							ExtVelocity[axisIdx]:= (newPos - OldPosition[axisIdx]) / (UDINT_TO_LREAL(_TaskInfo[1].CycleTime) / 10000000);
							OldPosition[axisIdx]:= newPos;
							ExtAcceleration :=  (ExtVelocity[axisIdx] - OldVelocity[axisIdx]) / (UDINT_TO_LREAL(_TaskInfo[1].CycleTime) / 10000000);
							OldVelocity[axisIdx]:= ExtVelocity[axisIdx];
							ExtDirection := SEL(newPos >= OldPosition[axisIdx], -1, 1);

							MC_ExtSetPointGenFeed(
								Position := newPos,
								Velocity := ExtVelocity[axisIdx],
								Acceleration := ExtAcceleration,
								Direction := ExtDirection,
								Axis := Axis[axisIdx].Axis);

						(*一般軸處理*)
						ELSE
							ExtVelocity[axisIdx]:= (TableOffsetPos[axisIdx] - OldPosition[axisIdx]) / (UDINT_TO_LREAL(_TaskInfo[1].CycleTime) / 10000000);
							OldPosition[axisIdx]:= TableOffsetPos[axisIdx];
							ExtAcceleration :=  (ExtVelocity[axisIdx] - OldVelocity[axisIdx]) / (UDINT_TO_LREAL(_TaskInfo[1].CycleTime) / 10000000);
							OldVelocity[axisIdx]:= ExtVelocity[axisIdx];
							ExtDirection := SEL(TableOffsetPos[axisIdx] >= OldPosition[axisIdx], -1, 1);
							//ExtDirection := SEL(TableOffsetPos[axisIdx] >= OldPosition[axisIdx], -1, 1);

							MC_ExtSetPointGenFeed(
								Position := TableOffsetPos[axisIdx],
								Velocity := ExtVelocity[axisIdx],
								Acceleration := ExtAcceleration,
								Direction := ExtDirection,
								Axis := Axis[axisIdx].Axis);
						END_IF
					END_IF
				END_FOR

				(* 目前送線動作結束 改idx*)
				IF AxisIsOn[FeederNo]
				AND CurrentTableIdx = FeederEndIdx[FeederIdx] + 1
				AND FeederEndIdx[FeederIdx] <> 0 THEN		

					FeederIdx := FeederIdx + 1;
					TouchOpenNo := 0;
					
				END_IF

				(* 探針動作結束 初始化 *)
				FOR touchIdx := 1 TO TouchNo DO

					IF CurrentTableIdx = TouchConfig[touchIdx].EndIdx[TouchConfigIdx[touchIdx]]
					AND TouchConfig[touchIdx].EndIdx[TouchConfigIdx[touchIdx]] <> 0 THEN
						IsTouch := FALSE;
						IsPreTouch := FALSE;
						TouchConfigIdx[touchIdx] := TouchConfigIdx[touchIdx] + 1;
					END_IF

					IF TouchConfigIdx[touchIdx] > 0 THEN
						IF CurrentTableIdx = TouchConfig[touchIdx].EndIdx[TouchConfigIdx[touchIdx] - 1] + 1
						AND TouchConfig[touchIdx].EndIdx[TouchConfigIdx[touchIdx] - 1] <> 0 THEN
							TouchMiss := FALSE;
						END_IF
					END_IF

				END_FOR

				(* 下一個探針動作的開始 先檢查是否探針前失誤 *)
								TouchPreCheck();

								NextCycleIdx();
				
								
				NextSubProgram();

			END_IF
	END_CASE

END_IF

ACTION AirFunc:

(*----------------Air----------------1,2,7,8是探針汽缸*)
(*非測試編輯時跑表*)
IF NOT (Inputstate.VRSwitch = FALSE AND State = ENUMSTATE.S_TEST) THEN
	FOR airIdx := 1 TO AirNo DO
		IF  airIdx <> 1 
		AND airIdx <> 2 
		AND airIdx <> 7
		AND airIdx <> 8 
		THEN
			AirIsOpen[airIdx] := AirTable[airIdx, CurrentTableIdx];
		END_IF
	END_FOR
END_IF
END_ACTION

ACTION CtrlSpeed:
IF Inputstate.ExFeederError
OR (IOSwitch.SaftyEnable AND 
        (Inputstate.SafetyError OR Inputstate.SafetyError1 OR Inputstate.SafetyError2 OR Inputstate.SafetyError3 OR Inputstate.SafetyError4) 
    ) 
THEN
    SpeedDownTo0 := TRUE;
    IF SpeedUPToOverride THEN
	    SpeedUPToOverride := FALSE;
        SpeedCtrlAccTimer(IN:=FALSE);
    END_IF
END_IF


IF lState <> State THEN
    lState := State;
    SpeedChanged := TRUE;
END_IF

IF SpeedUPToOverride THEN
	(*Reset Timer*)
	IF SpeedDownTo0 THEN
		SpeedDownTo0 := FALSE;
		SpeedCtrlDecTimer(IN:=FALSE);
	END_IF
    SpeedCtrlAccTimer(IN:=TRUE , PT:=SpeedAccDccTime , Q=> , ET=> );
    Speed        := Override * TIME_TO_REAL(SpeedCtrlAccTimer.ET) / TIME_TO_REAL(SpeedCtrlAccTimer.PT); (* 0 -> 1 *)
    IF SpeedCtrlAccTimer.Q THEN
        SpeedCtrlAccTimer(IN:=FALSE);
        SpeedUPToOverride := FALSE;
    END_IF
ELSIF SpeedDownTo0 THEN
    SpeedCtrlDecTimer(IN:=TRUE , PT:=SpeedAccDccTime , Q=> , ET=> );
    Speed        := Override * ( TIME_TO_REAL(SpeedCtrlDecTimer.PT) - TIME_TO_REAL(SpeedCtrlDecTimer.ET) ) / TIME_TO_REAL(SpeedCtrlDecTimer.PT); (* 1 -> 0 *)
ELSE
    IF SpeedChanged THEN
        IF LREAL_TO_DINT(Speed * 1000.0/100.0) = LREAL_TO_DINT(Override * 1000.0/100.0) THEN
            SpeedChanged := FALSE;
        ELSIF Speed < Override THEN
            Speed := Speed + 100.0/1000.0; (* 0->100% 用 1000ms *)
        ELSIF Speed > Override THEN
            Speed := Speed - 100.0/1000.0; (* 0->100% 用 1000ms *)
        END_IF
    ELSE
        Speed := Override;
    END_IF
END_IF
END_ACTION

ACTION EnableExtSetPoint:
	

FOR axisIdx := 1 TO No DO
	IF AxisIsOn[axisIdx] THEN
		Axis[axisIdx].EnableSetPointGenerator
		(
			Execute := TRUE,
			Position := Axis[axisIdx].ActPos,
			PositionType := POSITIONTYPE_ABSOLUTE,
			Axis :=  Axis[axisIdx].Axis
		);
	END_IF
END_FOR
ProduceState := S_WaitExtSetPoint;
END_ACTION

ACTION ExFeederFunc:

(*-------ExFeederSpeedUp------*)
IF State = ENUMSTATE.S_AUTO THEN
	ExFeederSpeedUp := ExFSpdUpTable[CurrentTableIdx];
END_IF
END_ACTION

ACTION FeederPosSetting:

FNeedHoldPos(
	IsTouch:= IsTouch,
	IsPreTouch := IsPreTouch,
	CurrentIdx:= CurrentTableIdx,
	FeederIdx	:= FeederIdx,
	FeederStartIdx:= FeederStartIdx,
	FeederEndIdx:=  FeederEndIdx,
	TouchConfig	    := TouchConfig,
	TouchConfigIdx := TouchConfigIdx,
 );

(* 計算位置 *)
IF FlashModeOn THEN

	IF(CurrentTableIdx = RepeatA) THEN
		(*閃電模式下，在A點是新的彈簧開始，根據offset進來次數不一定只會一次*)
		IF JumpFirstTime THEN
			JumpFirstTime := FALSE;
			Feeder.StillPos 	 := AxisTable1[axisIdx, FeederStartIdx[FeederIdx]] ;
			IF FNeedHoldPos.Yes = FALSE THEN
				Feeder.BasePos 	 := Feeder.CurPos - ( AxisTable1[axisIdx, RepeatA - 1] + ( AxisTable1[axisIdx, RepeatA] - AxisTable1[axisIdx, RepeatA - 1] ) * LastTableOffset );
			END_IF
		END_IF	
	ELSIF (CurrentTableIdx = JumpTiming) THEN
		IF JumpFirstTime THEN
			JumpFirstTime := FALSE;
			IF FNeedHoldPos.Yes = FALSE THEN
				Feeder.BasePos := Feeder.CurPos - ( AxisTable1[axisIdx, JumpTiming - 1] + ( AxisTable1[axisIdx, JumpTiming] - AxisTable1[axisIdx, JumpTiming - 1] ) * LastTableOffset );
			END_IF	
		END_IF
	END_IF

ELSIF CurrentTableIdx = G5Config[G5Status.CurIdx].ATime THEN

	IF G5Status.JumpFirstTime THEN
		G5Status.JumpFirstTime := FALSE;
		Feeder.StillPos 	 := AxisTable1[axisIdx, FeederStartIdx[FeederIdx]] ;	
		IF FNeedHoldPos.Yes = FALSE THEN
			Feeder.BasePos 	 := Feeder.CurPos - ( AxisTable1[axisIdx, CurrentTableIdx ]  );
		END_IF
	END_IF
	
END_IF

FSetCurPos();
END_ACTION

ACTION FeederVelAccSetting:
FNeedHoldPos(
	IsTouch:= IsTouch,
	IsPreTouch := IsPreTouch,
	CurrentIdx:= CurrentTableIdx,
	FeederIdx	:= FeederIdx,
	FeederStartIdx:= FeederStartIdx,
	FeederEndIdx:=  FeederEndIdx,
	TouchConfig	    := TouchConfig,
	TouchConfigIdx := TouchConfigIdx,
);
	
(*計算速度,加速度,方向*)
IF FNeedHoldPos.Yes THEN
	ExtVelocity[axisIdx]:= 0;
ELSE
	ExtVelocity[axisIdx]:= (Feeder.CurPos - OldPosition[axisIdx]) / (UDINT_TO_LREAL(_TaskInfo[1].CycleTime) / 10000000);
END_IF
OldPosition[axisIdx]:= Feeder.CurPos;
ExtDirection := SEL(Feeder.CurPos >= OldPosition[axisIdx], -1, 1);
ExtAcceleration :=  (ExtVelocity[axisIdx] - OldVelocity[axisIdx]) / (UDINT_TO_LREAL(_TaskInfo[1].CycleTime) / 10000000);
OldVelocity[axisIdx]:= ExtVelocity[axisIdx];
END_ACTION

ACTION FillAxisTable:
IF AxisTableBuf.OK THEN
	FOR axisIdx := 1 TO No DO
		FOR Idx := 0 TO 1999  DO
			AxisTable1[axisIdx, idx + SendOffset] := AxisTableBuf.Table[axisIdx, idx];
		END_FOR
	END_FOR
	SendOffset := SendOffset + 2000;
	AxisTableBuf.OK := FALSE;
	IF SendOffset >= TotalTimeByMs THEN
		SendOffset := 0;
		ProduceState := S_FillIOTable;
	END_IF
END_IF
IsGetTableBuf :=AxisTableBuf.OK;
END_ACTION

ACTION FillIOTable:

IsGetTableBuf := FALSE;
ReceiveAllBuf := TRUE;
IF TouchTableBuf.OK THEN
	TouchTableBuf.OK := FALSE;
	FOR touchIdx := 1 TO TouchNo DO
		FOR Idx := 0 TO 1999  DO
			TouchTable[touchIdx, idx + SendOffset] := TouchTableBuf.Table[touchIdx, idx];
		END_FOR
	END_FOR
	TouchTableFill := TRUE;
END_IF
IsGetTableBuf := IsGetTableBuf OR TouchTableFill;
ReceiveAllBuf := ReceiveAllBuf AND TouchTableFill;

IF AirTableBuf.OK THEN
	AirTableBuf.OK := FALSE;
	FOR airIdx := 1 TO AirNo DO
		FOR Idx := 0 TO 1999  DO
			AirTable[airIdx, idx + SendOffset] := AirTableBuf.Table[airIdx, idx];
		END_FOR
	END_FOR
	AirTableFill := TRUE;
END_IF
IsGetTableBuf := IsGetTableBuf OR AirTableFill;
ReceiveAllBuf := ReceiveAllBuf AND AirTableFill;

IF ExFSpdUpTableBuf.OK THEN
	ExFSpdUpTableBuf.OK := FALSE;
	FOR Idx := 0 TO 1999  DO
		ExFSpdUpTable[idx + SendOffset] := ExFSpdUpTableBuf.Table[idx];
	END_FOR
	ExFSpdUpTableFill := TRUE;
END_IF
IsGetTableBuf := IsGetTableBuf OR ExFSpdUpTableFill;
ReceiveAllBuf := ReceiveAllBuf AND ExFSpdUpTableFill;

IF ReceiveAllBuf THEN
	TouchTableFill := FALSE;
	AirTableFill := FALSE;
	ExFSpdUpTableFill := FALSE;
	SendOffset := SendOffset + 2000;
	IF SendOffset >= TotalTimeByMs THEN
		SendOffset := 0;
		ProduceState := S_FillSubTable;
	END_IF
END_IF
END_ACTION

ACTION FillSubIOTable:
IsGetTableBuf := FALSE;
IF SubProgramConfig[getSubNo].TotalTableSIze = 0 THEN
	ProduceState := S_FillTouchAdjustTable;
ELSE
    IF AirTableBuf.OK THEN
        FOR airIdx := 1 TO AirNo DO
            FOR Idx := 0 TO 1999  DO
                SubProgramTable[getSubNo].airTable[airIdx, idx + SendOffset] := AirTableBuf.Table[airIdx, idx];
            END_FOR
        END_FOR
        SendOffset := SendOffset + 2000;
        AirTableBuf.OK := FALSE;
        IF SendOffset >= SubProgramConfig[getSubNo].TotalTableSize THEN
            getSubNo := getSubNo + 1;
            SendOffset := 0;
        END_IF
    END_IF
    IsGetTableBuf := AirTableBuf.OK;
END_IF
END_ACTION

ACTION FillSubTable:

IsGetTableBuf := FALSE;
IF SubProgramConfig[getSubNo].TotalTableSIze = 0 THEN
	getSubNo := 1;
	ProduceState := S_FillSubIOTable;
ELSE
	IF AxisTableBuf.OK THEN
		FOR axisIdx := 1 TO No DO
			FOR Idx := 0 TO 1999  DO
				SubProgramTable[getSubNo].AxisTable[axisIdx, idx + SendOffset] := AxisTableBuf.Table[axisIdx, idx];
			END_FOR
		END_FOR
		SendOffset := SendOffset + 2000;
		AxisTableBuf.OK := FALSE;
		IF SendOffset >= SubProgramConfig[getSubNo].TotalTableSize THEN
			getSubNo := getSubNo + 1;
			SendOffset := 0;
		END_IF
	END_IF
	IsGetTableBuf := AxisTableBuf.OK;
END_IF
END_ACTION

ACTION FillTouchAdjustTable:
IsGetTableBuf := FALSE;
IF AxisTableBuf.OK THEN
    FOR axisIdx := 1 TO TouchAdjustNo DO
        IF TouchAdjustConfig[axisIdx].Enable THEN
            FOR idx := 0 TO 1999  DO
                TouchAdjustTable[axisIdx, idx + SendOffset] := AxisTableBuf.Table[axisIdx, idx];
            END_FOR
        END_IF        
    END_FOR
    SendOffset := SendOffset + 2000;
    AxisTableBuf.OK := FALSE;
    IF SendOffset >= TotalTimeByMs THEN
        SendOffset := 0;
        ProduceState := S_EnableExtSetPoint;
    END_IF
END_IF
IsGetTableBuf := AxisTableBuf.OK;
END_ACTION

ACTION FSetCurPos:

IF FNeedHoldPos.Yes THEN
	Feeder.CurPos := Feeder.BasePos + Feeder.TouchPos;
ELSE
	Feeder.CurPos := Feeder.BasePos + TableOffsetPos[axisIdx];
END_IF
END_ACTION

ACTION Initial:


FOR axisIdx:=1 TO No DO
	(*Set的最後一個點非0的時候沒清會爆衝*)
	Axis[axisIdx].Axis.PlcToNc.ExtSetPos := Axis[axisIdx].ActPos;
	Axis[axisIdx].EnableSetPointGenerator.Execute := FALSE;
	TableOffsetPos[axisIdx] := Axis[axisIdx].ActPos;
	OldPosition[axisIdx] := Axis[axisIdx].ActPos;
	OldVelocity[axisIdx] := 0;
	IsExtSetPointDone[axisIdx]:=FALSE;
	ModuloBase[axisIdx]  := Axis[axisIdx].ActPos;
END_FOR

ProFirstTime			:= FALSE;
Idx0FirstTime			:= TRUE;
ProduceState			:= S_FillAxisTable;
StartProNum				:= ProduceCurNum;
ProduceTimer			:= 0;
PPM						:= 0;
PPMCal(Clear := TRUE);
SpeedDownTo0			:= FALSE;
SpeedUPToOverride		:= FALSE;
SpeedCtrlAccTimer(IN:=FALSE);
SpeedCtrlDecTimer(IN:=FALSE);

JumpFirstTime		:= TRUE;

(*Send Table*)
getSubNo			:= 1;
SendOffset			:= 0;
TouchTableFill 		:= FALSE;
AirTableFill 			:= FALSE;
ExFSpdUpTableFill 	:= FALSE;

(*Index*)
CurrentTableIdx		:= 0;
CurrentTableOffset	:= 0;
LastTableOffset		:= 0;

(*IO*)
FOR touchIdx := 1 TO TouchNo DO
	TouchDist[touchIdx] 	 := 0;
	TouchConfigIdx[touchIdx] := 0;
	PreTouchShow[touchIdx]   := FALSE;
	ThisTurnTouchMissShow[touchIdx] := FALSE;
END_FOR
IsTouch				:= FALSE;
IsPreTouch			:= FALSE;
TouchOpenNo		:= 0;
TouchMiss			:= FALSE;
TouchBeforeStart		:= FALSE;
TouchMissNum		:= 0;
ThisTurnTouchMiss	:= FALSE;
IsOverUpBound		:= FALSE;
IsBelowDownBound	:= FALSE;
FeederIdx			:= 0;
Feeder.CurPos		:= Axis[FeederNo].Axis.NcToPlc.SetPos;
Feeder.BasePos	:= 0;
Feeder.StillPos		:= 0;
Feeder.TouchPos		:= 0;

AxisTableBuf.OK		:= FALSE;
TouchTableBuf.OK	:= FALSE;
AirTableBuf.OK		:= FALSE;
ExFSpdUpTableBuf.OK:= FALSE;

FOR TouchAdjustIdx := 1 TO TouchAdjustNo DO
	AdjustCounter[TouchAdjustIdx] := 0;
	AdjustCounterBuf[TouchAdjustIdx] := 0;
END_FOR

RunSubProgram		:= FALSE;
SubInFirstTime		:= TRUE;
RunSubNo			:=1;
SubTableIdx			:=0;
SubTableOffset		:=0;

(*油初始先開*)
FirstAutoRun := TRUE;

(*G5*)
G5Status.ATimeFIdx	   := 0;
G5Status.CurIdx		   := 1;
G5Status.CurTimes	   := 0;
G5Status.JumpFirstTime := FALSE;

lState	:= State;
SpeedChanged := FALSE;
END_ACTION

ACTION ModuloTurnsPlus1:
FOR axisIdx := 1 TO No DO
	IF AxesUseModulo[axisIdx] THEN
		AxesModuloTurns[axisIdx] := AxesModuloTurns[axisIdx] +  LREAL_TO_DINT( AxesModuloOGrad[axisIdx]) / AxesGradPerTurn[axisIdx];				
	END_IF
END_FOR
END_ACTION

ACTION NextCycleIdx:

(*探針失誤1次 設定也是一次 則 先暫停 => CurrentTableOffset 不變*)
IF TouchMissStop = FALSE THEN
	LastTableOffset := CurrentTableOffset;
	CurrentTableOffset := CurrentTableOffset + Speed/100;
END_IF

(*CurrentTableIdx增加的時候*)
IF CurrentTableOffset >= 1 THEN
	CurrentTableOffset := CurrentTableOffset - 1;
	(*閃電模式*)
	IF FlashModeOn THEN
		(*RepeatA*)
		IF CurrentTableIdx = RepeatA THEN
			(*紀錄RepeatA時的FeederIdx給跳回來時設定*)
			RepeatA_FeederIdx 	:= FeederIdx;
			FOR touchIdx := 1 TO TouchNo DO
				RepeatA_TouchConfigIdx[touchIdx] := TouchConfigIdx[touchIdx];
			END_FOR
			CurrentTableIdx 	:= CurrentTableIdx + 1;
			(*第一條*)
			IF StartProNum = ProduceCurNum THEN
								ModuloTurnsPlus1();
				ProduceCurNum	:= ProduceCurNum + 1;
				PPMCal( CurTime := ProduceTimer, PPM => PPM );
				IF ProduceCurNum = ProduceNum THEN(*無法停止已經做到一半必須做完*)
					ProduceNum	:= ProduceNum + 1;
				END_IF
			END_IF
		(*RepeatB*)
	 	ELSIF CurrentTableIdx = RepeatB THEN
			IF ProduceCurNum < ProduceNum - 1 THEN
				JumpFirstTime 	:= TRUE;
				CurrentTableIdx := RepeatA;
				FeederIdx		:= RepeatA_FeederIdx;	
				FOR touchIdx := 1 TO TouchNo DO
					TouchConfigIdx[touchIdx] := RepeatA_TouchConfigIdx[touchIdx];
				END_FOR
				FOR axisIdx := 1 TO No DO
					IF AxesUseModulo[axisIdx] THEN
						ModuloBase[axisIdx] := ModuloBase[axisIdx] + AxesModuloOGrad[axisIdx];
					END_IF
				END_FOR	
								ModuloTurnsPlus1();
				ProduceCurNum 	:= ProduceCurNum + 1;
				PPMCal( CurTime := ProduceTimer, PPM => PPM );
			ELSIF ProduceCurNum = ProduceNum - 1 THEN
								ModuloTurnsPlus1();
				ProduceNum		:= ProduceNum + 1;(*無法停止已經做到一半必須做完*)
				ProduceCurNum 	:= ProduceCurNum + 1;
				PPMCal( CurTime := ProduceTimer, PPM => PPM );
				CurrentTableIdx := CurrentTableIdx + 1;
			ELSE
				CurrentTableIdx := CurrentTableIdx + 1;
			END_IF
		(*停機時機1*)	(*停機時機2*)
		ELSIF CurrentTableIdx = StopTiming1 OR CurrentTableIdx = StopTiming2 THEN

			IF ProduceCurNum = ProduceNum - 1 THEN

				IF CurrentTableIdx = StopTiming1 THEN
					FOR axisIdx := 1 TO No DO
						IF AxesUseModulo[axisIdx] THEN
							ModuloBase[axisIdx] := ModuloBase[axisIdx] - 2 * AxesModuloOGrad[axisIdx];
						END_IF
					END_FOR		
				ELSIF CurrentTableIdx = StopTiming2 THEN
					FOR axisIdx := 1 TO No DO
						IF AxesUseModulo[axisIdx] THEN
							ModuloBase[axisIdx] := ModuloBase[axisIdx] - AxesModuloOGrad[axisIdx];
						END_IF
					END_FOR	
				END_IF

				CurrentTableIdx 	 := JumpTiming;
				JumpFirstTime		 := TRUE;

			(*探針停機*)
			ELSIF TouchMissNum = TouchMissSetNum AND TouchMissSetNum <> 0 THEN		
								ModuloTurnsPlus1();
				ProduceNum 			 := ProduceCurNum + 1;
				CurrentTableIdx 	 := JumpTiming;
				JumpFirstTime		 := TRUE;
				
			ELSE
				(*下條彈簧開始*)
				FOR touchIdx := 1 TO TouchNo DO
					TouchDist[touchIdx] := 0;
				END_FOR
				CurrentTableIdx 	 := CurrentTableIdx + 1;
			END_IF
		ELSE
			CurrentTableIdx 	 := CurrentTableIdx + 1;
		END_IF
		
	ELSIF CurrentTableIdx = G5Config[G5Status.CurIdx].ATime THEN
		CurrentTableIdx    := CurrentTableIdx + 1;
		G5Status.ATimeFIdx := FeederIdx;
		G5Status.ATimeSubNo:= RunSubNo;
		FOR touchIdx := 1 TO TouchNo DO
			G5Status.ATimeTouchConfigIdx[touchIdx] := TouchConfigIdx[touchIdx];
		END_FOR

	ELSIF CurrentTableIdx = G5Config[G5Status.CurIdx].BTime AND G5Status.CurTimes < G5Config[G5Status.CurIdx].RepeatTimes THEN
		CurrentTableIdx 	   := G5Config[G5Status.CurIdx].ATime;
		FeederIdx			   := G5Status.ATimeFIdx;
		RunSubNo 			   := G5Status.ATimeSubNo;
		G5Status.JumpFirstTime := TRUE;
		G5Status.CurTimes	   := G5Status.CurTimes + 1;
		IsHookMovable			   := FALSE;
		FOR touchIdx := 1 TO TouchNo DO
			TouchConfigIdx[touchIdx] := G5Status.ATimeTouchConfigIdx[touchIdx];
		END_FOR

	ELSIF CurrentTableIdx = G5Config[G5Status.CurIdx].BTime AND G5Status.CurTimes = G5Config[G5Status.CurIdx].RepeatTimes THEN
		IF G5Config[G5Status.CurIdx].BTime = G5Config[G5Status.CurIdx + 1].ATime AND G5Status.CurIdx + 1 <= G5ConfigNo THEN
			G5Status.ATimeFIdx := FeederIdx;
			G5Status.ATimeSubNo:= RunSubNo;
			FOR touchIdx := 1 TO TouchNo DO
				G5Status.ATimeTouchConfigIdx[touchIdx] := TouchConfigIdx[touchIdx];
			END_FOR
		END_IF
		CurrentTableIdx   := CurrentTableIdx + 1;
		G5Status.CurIdx   := G5Status.CurIdx + 1;
		G5Status.CurTimes := 0;
		IsHookMovable		  := TRUE;
	ELSE
	(*一般情況*)
		CurrentTableIdx := CurrentTableIdx + 1;
	END_IF
END_IF

IF CurrentTableIdx = TotalTimeByMs THEN
	(*到達探針失誤量就停機*)
	IF TouchMissNum >= TouchMissSetNum AND TouchMissSetNum <> 0 THEN
	 	ProduceNum := ProduceCurNum;
	ELSE		
		CurrentTableIdx 	:= 0;
		RunSubNo			:= 1;
		G5Status.CurIdx		:= 1;
		G5Status.CurTimes	:= 0;
		Idx0FirstTime		:= TRUE;
				ModuloTurnsPlus1();
		ProduceCurNum   := ProduceCurNum + 1;
		PPMCal( CurTime := ProduceTimer, PPM => PPM );
	END_IF
END_IF
END_ACTION

ACTION NextSubProgram:

(*切換到下個副程式*)
IF RunSubNo <= SubProgramNo
AND SubProgramConfig[RunSubNo].TotalTableSize <> 0
AND CurrentTableIdx > SubProgramConfig[RunSubNo].EndIdx + 1 THEN
	RunSubNo := RunSubNo + 1;
END_IF
END_ACTION

ACTION OilFunc:
FOR idx := 1 TO OilNo DO
	IF Oil[idx].Enable THEN

	(*要初始化
	Oil[idx].IsOpen := TRUE;
	Oil[idx].CurTime := 0;
	Oil[idx].CurStrokes := 0;
	OilStrokeCount[idx] := ProduceCurNum;
	*)

		IF Oil[idx].IsOpen THEN
			IF Oil[idx].OpenTime <> 0 AND Oil[idx].CurTime < Oil[idx].OpenTime THEN
				Oil[idx].CurTime := Oil[idx].CurTime + 1;
				IF Oil[idx].CurTime >= Oil[idx].OpenTime THEN
					Oil[idx].CurTime :=0;
					Oil[idx].IsOpen := FALSE;
					OilStrokeCount[idx] := ProduceCurNum;
				END_IF
			END_IF
		ELSE
			IF Oil[idx].CloseTime <> 0 AND Oil[idx].CurTime < Oil[idx].CloseTime THEN
				Oil[idx].CurTime := Oil[idx].CurTime + 1;
				IF Oil[idx].CurTime >= Oil[idx].CloseTime THEN
					Oil[idx].CurTime :=0;
					Oil[idx].IsOpen := TRUE;
				END_IF
			ELSIF Oil[idx].CloseStrokes <> 0 AND Oil[idx].CurStrokes <= Oil[idx].CloseStrokes
			AND OilStrokeCount[idx] <> ProduceCurNum
			THEN
				OilStrokeCount[idx] := ProduceCurNum;
				Oil[idx].CurStrokes := Oil[idx].CurStrokes + 1;
				IF Oil[idx].CurStrokes = Oil[idx].CloseStrokes THEN (*當下那圈不算*)
					Oil[idx].CurStrokes :=0;
					Oil[idx].IsOpen := TRUE;
				END_IF
			END_IF
		END_IF

	ELSE
		Oil[idx].IsOpen := FALSE;
	END_IF
END_FOR
END_ACTION

ACTION SubAirFunc:
(*----------------SubAir----------------1,2,7,8是探針汽缸*)
(*非測試編輯時跑表*)
IF NOT (Inputstate.VRSwitch = FALSE AND State = ENUMSTATE.S_TEST) THEN
	FOR airIdx := 1 TO AirNo DO
		IF  airIdx <> 1 
		AND airIdx <> 2 
		AND airIdx <> 7 
		AND airIdx <> 8 
		THEN
			AirIsOpen[airIdx] := SubProgramTable[RunSubNo].AirTable[airIdx, SubTableIdx];
		END_IF
	END_FOR
END_IF
END_ACTION

ACTION TouchFunc:

FOR touchIdx := 1 TO TouchNo DO

	(* 還沒開始就探到 探針失誤 StartIdx *)
	IF CurrentTableIdx = TouchConfig[touchIdx].StartIdx[TouchConfigIdx[touchIdx]]
	 AND TouchConfig[touchIdx].StartIdx[TouchConfigIdx[touchIdx]] <> TouchConfig[touchIdx].EndIdx[TouchConfigIdx[touchIdx]]
	 AND DigInSlave[2].Input[touchIdx] AND NOT TouchMiss THEN

		IsPreTouch			:= TRUE;
		PreTouchShow[touchIdx]   := TRUE;
		ThisTurnTouchMissShow[touchIdx]   := FALSE;
		TouchMiss 			:= TRUE;
		ThisTurnTouchMiss   := TRUE;
		TouchMissNum 		:= TouchMissNum + 1;
		IsTouchWithF 		:= FALSE;

		(*到達失誤量*)
		IF TouchMissNum = TouchMissSetNum AND TouchMissSetNum = 1 THEN
			(*一次直接Error Reset*)
			TouchMissStop := TRUE;
		END_IF
		(*有送線*)
		IF CurrentTableIdx = FeederStartIdx[FeederIdx] OR CurrentTableIdx = FeederEndIdx[FeederIdx] THEN

			TableOffsetPos[FeederNo]:= AxisTable1[FeederNo, CurrentTableIdx];

			Feeder.TouchPos 		:= TableOffsetPos[FeederNo];
			Feeder.TouchFeederIdx 	:= FeederIdx;
			TouchDist[touchIdx] 	:= 0;
			FTouchShowPos 			:= 0;
			IsTouchWithF 		:= TRUE;

		ELSE
			TouchDist[touchIdx]		:= 0;
			FTouchShowPos			:= TouchDist[touchIdx];
		END_IF

	(* 探針中 StartIdx+1 ~ EndIdx-1 *)
	ELSIF CurrentTableIdx > TouchConfig[touchIdx].StartIdx[TouchConfigIdx[touchIdx]]
	  AND CurrentTableIdx < TouchConfig[touchIdx].EndIdx[TouchConfigIdx[touchIdx]]
	  AND DigInSlave[2].Input[touchIdx] AND NOT TouchMiss AND NOT IsPreTouch AND NOT IsTouch THEN

		IsTouch := TRUE;
		TouchOpenNo	:= touchIdx;
		IsTouchWithF 		:= FALSE;

		(* 有送線 送線開啟*)
		IF AxisIsOn[FeederNo]
		AND (CurrentTableIdx > FeederStartIdx[FeederIdx]
		AND  CurrentTableIdx < FeederEndIdx[FeederIdx]) THEN	

			Feeder.TouchPos := TableOffsetPos[FeederNo];
			Feeder.TouchFeederIdx := FeederIdx;
			TouchDist[touchIdx] := Feeder.TouchPos - Feeder.StillPos;
			FTouchShowPos := TouchDist[touchIdx];
			IsTouchWithF 		:= TRUE;

			(* 探針補償 *)
			IsAdjustTouch(touchNo := touchIdx, CurrentTableIdx := CurrentTableIdx);
			IF IsAdjustTouch.Yes THEN

				(* 在公差範圍外算是失誤 *)
				IF TouchDist[touchIdx] < TouchAdjustConfig[IsAdjustTouch.AdjustIdx].DownBound 
				OR TouchDist[touchIdx] > TouchAdjustConfig[IsAdjustTouch.AdjustIdx].UpBound THEN

					IF TouchDist[touchIdx] < TouchAdjustConfig[IsAdjustTouch.AdjustIdx].DownBound THEN
						PreTouchShow[touchIdx]   := TRUE;
						IsBelowDownBound := TRUE;
					ELSE
						ThisTurnTouchMissShow[touchIdx] := TRUE;
						IsOverUpBound := TRUE;
					END_IF

					TouchMiss 			:= TRUE;
					ThisTurnTouchMiss   := TRUE;
					TouchMissNum 		:= TouchMissNum + 1;

					(*到達失誤量*)
					IF TouchMissNum = TouchMissSetNum AND TouchMissSetNum = 1 THEN
						(*一次直接Error Reset*)
						TouchMissStop := TRUE;
					END_IF
				
				ELSIF TouchDist[touchIdx] > TouchAdjustConfig[IsAdjustTouch.AdjustIdx].RangeUp THEN
					IF AdjustCounter[IsAdjustTouch.AdjustIdx] + 1 <= TouchAdjustConfig[IsAdjustTouch.AdjustIdx].UpCountLimit THEN (* 4 + 1 <= 5.5 *)

						AdjustCounterBuf[IsAdjustTouch.AdjustIdx] := AdjustCounterBuf[IsAdjustTouch.AdjustIdx] + 1;

					ELSIF AdjustCounter[IsAdjustTouch.AdjustIdx] + 1 - TouchAdjustConfig[IsAdjustTouch.AdjustIdx].UpCountLimit < 1 THEN (*5 + 1 - 5.5 < 1*)

						AdjustCounterBuf[IsAdjustTouch.AdjustIdx] := TouchAdjustConfig[IsAdjustTouch.AdjustIdx].UpCountLimit - AdjustCounter[IsAdjustTouch.AdjustIdx];(* 5.5 - 5 *)
					END_IF

				ELSIF TouchDist[touchIdx] < TouchAdjustConfig[IsAdjustTouch.AdjustIdx].RangeDown THEN
					IF AdjustCounter[IsAdjustTouch.AdjustIdx] - 1 >= TouchAdjustConfig[IsAdjustTouch.AdjustIdx].DownCountLimit THEN (* -4 - 1 >= -5.5 *)

						AdjustCounterBuf[IsAdjustTouch.AdjustIdx] := AdjustCounterBuf[IsAdjustTouch.AdjustIdx] - 1;

					ELSIF AdjustCounter[IsAdjustTouch.AdjustIdx] - 1 - TouchAdjustConfig[IsAdjustTouch.AdjustIdx].DownCountLimit > -1 THEN (* -5 - 1 - (-5.5) > -1  *)

						AdjustCounterBuf[IsAdjustTouch.AdjustIdx] := TouchAdjustConfig[IsAdjustTouch.AdjustIdx].DownCountLimit - AdjustCounter[IsAdjustTouch.AdjustIdx];(* -5.5 - (-5) *)

					END_IF

				END_IF

			END_IF

		ELSE
			TouchDist[touchIdx]		:= 0;
			FTouchShowPos			:= TouchDist[touchIdx];
		END_IF

	(* 探針結束還沒探到 探針失誤 EndIdx *)
	ELSIF CurrentTableIdx = TouchConfig[touchIdx].EndIdx[TouchConfigIdx[touchIdx]]
      AND TouchConfig[touchIdx].EndIdx[TouchConfigIdx[touchIdx]] <> 0
	  AND NOT IsTouch AND NOT TouchMiss THEN

		TouchMiss := TRUE;
		TouchDist[TouchOpenNo] := 0;
		TouchMissNum := TouchMissNum + 1;
		ThisTurnTouchMiss	:= TRUE;
		PreTouchShow[touchIdx]   := FALSE;
		ThisTurnTouchMissShow[touchIdx] := TRUE;
		(*到達失誤量*)
		IF TouchMissNum = TouchMissSetNum AND TouchMissSetNum = 1 THEN
			(*一次直接Error Reset*)
			TouchMissStop := TRUE;
		END_IF


	(* 有開啟全域探針 *)
	ELSIF IOSwitch.GlobalTouchEnable THEN

		InAnotherTouch(CurrTouchIdx:=touchIdx, CurrentIdx:=CurrentTableIdx, TouchConfig:=TouchConfig, TouchConfigIdx:=TouchConfigIdx);
		(* 除了探針動作之外碰到 算是探針異常 *)
		IF NOT InAnotherTouch.Yes
		AND CurrentTableIdx < TouchConfig[touchIdx].StartIdx[TouchConfigIdx[touchIdx]]
		AND TouchConfig[touchIdx].StartIdx[TouchConfigIdx[touchIdx]] <> TouchConfig[touchIdx].EndIdx[TouchConfigIdx[touchIdx]]
		AND DigInSlave[2].Input[touchIdx] AND NOT TouchMiss THEN

			TouchMiss 			:= TRUE;
			ThisTurnTouchMiss	:= TRUE;
			PreTouchShow[touchIdx]   := FALSE;
			ThisTurnTouchMissShow[touchIdx] := FALSE;
			GlobalTouchShow[touchIdx]     := TRUE;
			TouchMissNum 		:= TouchMissNum + 1;
			(*到達失誤量*)
			IF TouchMissNum = TouchMissSetNum AND TouchMissSetNum = 1 THEN
				(*一次直接Error Reset*)
				TouchMissStop := TRUE;
			END_IF

		(* 探針前已經失誤 設定IsPreTouch 不要送線*)
		ELSIF CurrentTableIdx = TouchConfig[touchIdx].StartIdx[TouchConfigIdx[touchIdx]]
		AND TouchConfig[touchIdx].StartIdx[TouchConfigIdx[touchIdx]] <> TouchConfig[touchIdx].EndIdx[TouchConfigIdx[touchIdx]]
		AND TouchMiss THEN

			IsPreTouch			:= TRUE;
			PreTouchShow[touchIdx]   := FALSE;
			ThisTurnTouchMissShow[touchIdx] := FALSE;
			GlobalTouchShow[touchIdx]     := TRUE;
			IsTouchWithF 		:= FALSE;

			(*有送線*)
			IF CurrentTableIdx = FeederStartIdx[FeederIdx] OR CurrentTableIdx = FeederEndIdx[FeederIdx] THEN

				TableOffsetPos[FeederNo]:= AxisTable1[FeederNo, CurrentTableIdx];

				Feeder.TouchPos 		:= TableOffsetPos[FeederNo];
				Feeder.TouchFeederIdx 	:= FeederIdx;
				TouchDist[touchIdx] 	:= 0;
				FTouchShowPos 			:= 0;
				IsTouchWithF 		:= TRUE;

			ELSE
				TouchDist[touchIdx]		:= 0;
				FTouchShowPos			:= TouchDist[touchIdx];
			END_IF
		END_IF

	END_IF

END_FOR

(*----------------Touch Air----------------*)
(*非測試編輯時跑表*)
IF NOT (Inputstate.VRSwitch = FALSE AND State = ENUMSTATE.S_TEST) THEN
	FOR touchIdx := 1 TO TouchNo DO
		IF IsTouch OR TouchMiss
		OR TouchConfigIdx[touchIdx] > 0 AND CurrentTableIdx = TouchConfig[touchIdx].EndIdx[TouchConfigIdx[touchIdx]]
		//		OR TouchConfigIdx[touchIdx] > 0 AND CurrentTableIdx = TouchConfig[touchIdx].EndIdx[TouchConfigIdx[touchIdx] - 1]
		OR CurrentTableIdx = TouchConfig[touchIdx].EndIdx[TouchConfigIdx[touchIdx]] AND TouchConfig[touchIdx].EndIdx[TouchConfigIdx[touchIdx]] <> 0 THEN
			IF touchIdx = 3 THEN
				AirIsOpen[7] := FALSE;
			ELSIF touchIdx = 4 THEN
				AirIsOpen[8] := FALSE;
			ELSE
				AirIsOpen[touchIdx] := FALSE;
			END_IF
		ELSE
			IF touchIdx = 3 THEN
				AirIsOpen[7] := AirTable[7, CurrentTableIdx];
			ELSIF touchIdx = 4 THEN
				AirIsOpen[8] := AirTable[8, CurrentTableIdx];
			ELSE
				AirIsOpen[touchIdx] := AirTable[touchIdx, CurrentTableIdx];
			END_IF
		END_IF
	END_FOR
END_IF
END_ACTION

ACTION TouchPreCheck:

FOR touchIdx := 1 TO TouchNo DO

	(* 還沒開始就探到 探針失誤 StartIdx *)
	IF CurrentTableIdx = TouchConfig[touchIdx].StartIdx[TouchConfigIdx[touchIdx]]
	 AND TouchConfig[touchIdx].StartIdx[TouchConfigIdx[touchIdx]] <> TouchConfig[touchIdx].EndIdx[TouchConfigIdx[touchIdx]]
	 AND DigInSlave[2].Input[touchIdx] AND NOT TouchMiss THEN			 

		IsPreTouch			:= TRUE;
		PreTouchShow[touchIdx]   := TRUE;
		ThisTurnTouchMissShow[touchIdx]   := FALSE;
		TouchMiss 			:= TRUE;
		ThisTurnTouchMiss   := TRUE;
		TouchMissNum 		:= TouchMissNum + 1;
		IsTouchWithF 		:= FALSE;

		(*到達失誤量*)
		IF TouchMissNum = TouchMissSetNum AND TouchMissSetNum = 1 THEN
			(*一次直接Error Reset*)
			TouchMissStop := TRUE;
		END_IF
		(*有送線*)
		IF CurrentTableIdx = FeederStartIdx[FeederIdx] OR CurrentTableIdx = FeederEndIdx[FeederIdx] THEN

			TableOffsetPos[FeederNo]:= AxisTable1[FeederNo, CurrentTableIdx];

			Feeder.TouchPos 		:= TableOffsetPos[FeederNo];
			Feeder.TouchFeederIdx 	:= FeederIdx;
			TouchDist[touchIdx] 	:= 0;
			FTouchShowPos 			:= 0;
			IsTouchWithF 		:= TRUE;

		ELSE
			TouchDist[touchIdx]		:= 0;
			FTouchShowPos			:= TouchDist[touchIdx];
		END_IF
		
	END_IF
END_FOR
END_ACTION

ACTION WaitExtSetPoint:


IsSetPointComplete := TRUE;
FOR axisIdx := 1 TO No DO
	IF AxisIsOn[axisIdx] THEN
		IF Axis[axisIdx].EnableSetPointGenerator.Done THEN
			Axis[axisIdx].EnableSetPointGenerator.Execute := FALSE;
			IsExtSetPointDone[axisIdx] := TRUE;
		END_IF
		IsSetPointComplete := IsSetPointComplete AND IsExtSetPointDone[axisIdx];
	END_IF
END_FOR
IF IsSetPointComplete THEN
	ProduceState := S_Run;
END_IF
END_ACTION

END_PROGRAM

// ---- POUs/FB/FB_CloseIO.TcPOU
FUNCTION_BLOCK FB_CloseIO
VAR_INPUT
END_VAR
VAR_OUTPUT
END_VAR
VAR
	idx				: INT:=1;
	CloseAir			: FB_CloseAir;
	CloseOil			: FB_CloseOil;
END_VAR

FOR idx:=1 TO TouchNo DO
	Touch[idx].CurTime := 0;
END_FOR

CloseAir();

CloseOil();

END_FUNCTION_BLOCK

// ---- POUs/FB/FB_CloseAir.TcPOU
FUNCTION_BLOCK FB_CloseAir
VAR_INPUT
END_VAR
VAR_OUTPUT
END_VAR
VAR
	idx				: INT:=1;
END_VAR


FOR idx:= 1 TO AirNo DO
	AirIsOpen[idx] := FALSE;
END_FOR

END_FUNCTION_BLOCK

// ---- POUs/FB/PPMCal.TcPOU
FUNCTION_BLOCK PPMCal
VAR_INPUT
	Clear	: BOOL;
	CurTime  : UDINT;
END_VAR
VAR_OUTPUT
	PPM	:REAL;
END_VAR
VAR
	OrigTime:UDINT;
END_VAR

IF Clear THEN
	Clear 	:= FALSE;
	PPM	:=  0;
	OrigTime := 0;
ELSE
	PPM := 1000.0/UDINT_TO_REAL(CurTime - OrigTIme) * 60.0;
	OrigTIme := CurTime;
END_IF

END_FUNCTION_BLOCK

// ---- POUs/FB/FB_FNeedHoldPos.TcPOU
FUNCTION_BLOCK FB_FNeedHoldPos
VAR_INPUT
	IsTouch			: BOOL;
	IsPreTouch		: BOOL;
	CurrentIdx		: DINT;
	FeederStartIdx	: ARRAY [0..999] OF DINT;
	FeederEndIdx	: ARRAY [0..999] OF DINT;
	FeederIdx		: INT := 0;
	TouchConfig		: ARRAY [1..TouchNo] OF ST_TouchConfig;
	TouchConfigIdx	: ARRAY [1..TouchNo] OF  INT;
END_VAR
VAR_OUTPUT
	Yes				:BOOL;
END_VAR
VAR
	touchIdx			:INT;
END_VAR


Yes := FALSE;

IF (IsTouch AND CurrentIdx > FeederStartIdx[FeederIdx]  AND  CurrentIdx < FeederEndIdx[FeederIdx]) THEN
	Yes := TRUE;
ELSIF IsPreTouch THEN
	FOR touchIdx := 1 TO TouchNo DO
		IF    CurrentIdx >= TouchConfig[touchIdx].StartIdx[TouchConfigIdx[touchIdx]] AND CurrentIdx < TouchConfig[touchIdx].EndIdx[TouchConfigIdx[touchIdx]]
		OR CurrentIdx >= TouchConfig[touchIdx].StartIdx[TouchConfigIdx[touchIdx] + 1] AND CurrentIdx < TouchConfig[touchIdx].EndIdx[TouchConfigIdx[touchIdx] + 1] THEN
			Yes := TRUE;
		END_IF
	END_FOR
END_IF

END_FUNCTION_BLOCK

// ---- POUs/FB/FB_TouchEnd.TcPOU
FUNCTION_BLOCK FB_TouchEnd
VAR_INPUT
	CurrentIdx		: DINT;
	TouchConfig		: ARRAY [1..TouchNo] OF ST_TouchConfig;
	TouchConfigIdx	: ARRAY [1..TouchNo] OF  INT;
END_VAR
VAR_OUTPUT
	Yes				:BOOL;
END_VAR
VAR
	touchIdx			:INT;
END_VAR


Yes := FALSE;

FOR touchIdx := 1 TO TouchNo DO
	IF CurrentIdx = TouchConfig[touchIdx].EndIdx[TouchConfigIdx[touchIdx]]
    AND TouchConfig[touchIdx].EndIdx[TouchConfigIdx[touchIdx]] <> 0
	THEN
		Yes := TRUE;
	END_IF
END_FOR

END_FUNCTION_BLOCK

// ---- POUs/FB/FB_InAnotherTouch.TcPOU
FUNCTION_BLOCK FB_InAnotherTouch
VAR_INPUT
	CurrTouchIdx	: INT;
	CurrentIdx		: DINT;
	TouchConfig		: ARRAY [1..TouchNo] OF ST_TouchConfig;
	TouchConfigIdx	: ARRAY [1..TouchNo] OF  INT;
END_VAR
VAR_OUTPUT
	Yes				:BOOL;
END_VAR
VAR
	touchIdx			:INT;
END_VAR


Yes := FALSE;

FOR touchIdx := 1 TO TouchNo DO
	IF touchIdx <> CurrTouchIdx
	AND CurrentIdx > TouchConfig[touchIdx].StartIdx[TouchConfigIdx[touchIdx]]
	AND CurrentIdx < TouchConfig[touchIdx].EndIdx[TouchConfigIdx[touchIdx]] THEN
		Yes := TRUE;
	END_IF
END_FOR

END_FUNCTION_BLOCK

// ---- POUs/FB/FB_IsAdjustAxis.TcPOU
FUNCTION_BLOCK FB_IsAdjustAxis
VAR_INPUT
	pAxis			:INT;
	CurrentTableIdx :DINT;
END_VAR
VAR_OUTPUT
	Yes				:BOOL;
	AdjustIdx		:INT;
END_VAR
VAR
	touchAdjustIdx	:INT;
END_VAR

AdjustIdx := -1;
FOR touchAdjustIdx := 1 TO TouchAdjustNo DO
	IF TouchAdjustConfig[TouchAdjustIdx].Enable AND pAxis = TouchAdjustConfig[TouchAdjustIdx].pAxis 
	AND CurrentTableIdx >= TouchAdjustConfig[TouchAdjustIdx].AdjustStartIdx AND CurrentTableIdx <= TouchAdjustConfig[TouchAdjustIdx].AdjustEndIdx
	THEN
		AdjustIdx := TouchAdjustIdx;
	END_IF
END_FOR
IF AdjustIdx <> -1 THEN
	Yes := TRUE;
ELSE
	Yes := FALSE;
END_IF

END_FUNCTION_BLOCK

// ---- POUs/FB/FB_IsAdjustTouch.TcPOU
FUNCTION_BLOCK FB_IsAdjustTouch
VAR_INPUT
	touchNo			:INT;
	CurrentTableIdx :DINT;
END_VAR
VAR_OUTPUT
	Yes				:BOOL;
	AdjustIdx		:INT;
END_VAR
VAR
	touchAdjustIdx	:INT;
END_VAR


AdjustIdx := -1;
FOR touchAdjustIdx := 1 TO TouchAdjustNo DO
	IF TouchAdjustConfig[TouchAdjustIdx].Enable AND touchNo = TouchAdjustConfig[TouchAdjustIdx].TouchNo
	AND CurrentTableIdx >= TouchAdjustConfig[TouchAdjustIdx].TouchStartIdx AND CurrentTableIdx <= TouchAdjustConfig[TouchAdjustIdx].TouchEndIdx THEN
		AdjustIdx := TouchAdjustIdx;
	END_IF
END_FOR
IF AdjustIdx <> -1 THEN
	Yes := TRUE;
ELSE
	Yes := FALSE;
END_IF

END_FUNCTION_BLOCK

// ---- POUs/SubRunAlone.TcPOU
PROGRAM SubRunAlone
VAR
   	SubRunAloneState :(S_FillSubTable, S_FillSubIOTable,  S_EnableExtSetPoint, S_WaitExtSetPoint, S_Run, S_Complete);
	IsAutoRun 			:BOOL;
	Idx0FirstTime			:BOOL;
	idx					:INT ;
	axisIdx				:INT;
    airIdx				:INT;
	SendOffset			:UDINT := 0;
	RunSubNo			:INT;
	SubSpeed			:REAL:= 30;
	CurrentTableIdx		:DINT;
	CurrentTableOffset	:REAL;

	IsExtSetPointDone		:ARRAY [1..No] OF BOOL;
	IsSetPointComplete 	:BOOL;
	TableOffsetPos		:ARRAY [1..No] OF  LREAL;
	OldPosition			:ARRAY [1..No] OF LREAL;
	ExtVelocity			:ARRAY [1..No] OF LREAL;
	OldVelocity			:ARRAY [1..No] OF LREAL;
	ExtAcceleration		:LREAL;
	ExtDirection			:DINT;
END_VAR


IF SubRunning THEN

	IF SubRunAloneFirstTime THEN
		(*初始化*)
				Initial();
	END_IF

	CASE SubRunAloneState OF

		S_FillSubTable:
						FillSubTable();

		S_FillSubIOTable:
						FillSubIOTable();

		S_EnableExtSetPoint:
						EnableExtSetPoint();

		S_WaitExtSetPoint:
						WaitExtSetPoint();

		S_Run:

			(* 表一開始 初始*)
			IF CurrentTableIdx = 0 AND Idx0FirstTime THEN
				Idx0FirstTime 		:= FALSE;
				OldPosition[axisIdx] 	:= 0;
				OldVelocity[axisIdx] 	:= 0;
			END_IF



			(*副程式*)

			(* 設定ExtPosition *)
			FOR axisIdx := 1 TO No DO
				IF AxisIsOn[axisIdx] THEN
					(* 超過這條最後idx *)
					IF (CurrentTableIdx + CurrentTableOffset) > (SubProgramConfig[RunSubNo].TotalTableSize - 1) THEN
						TableOffsetPos[axisIdx]:= SubProgramTable[RunSubNo].AxisTable[axisIdx, CurrentTableIdx];
					ELSE
					(* idx在此表內 *)
						TableOffsetPos[axisIdx]:= SubProgramTable[RunSubNo].AxisTable[axisIdx, CurrentTableIdx] + ( SubProgramTable[RunSubNo].AxisTable[axisIdx, CurrentTableIdx + 1] - SubProgramTable[RunSubNo].AxisTable[axisIdx, CurrentTableIdx] ) * CurrentTableOffset;
					END_IF
				END_IF
			END_FOR

						SubAirFunc();

			FOR axisIdx := 1 TO No DO
				IF AxisIsOn[axisIdx] THEN
					ExtVelocity[axisIdx]:= (TableOffsetPos[axisIdx] - OldPosition[axisIdx]) / (UDINT_TO_LREAL(_TaskInfo[1].CycleTime) / 10000000);
					OldPosition[axisIdx]:= TableOffsetPos[axisIdx];
					ExtAcceleration :=  (ExtVelocity[axisIdx] - OldVelocity[axisIdx]) / (UDINT_TO_LREAL(_TaskInfo[1].CycleTime) / 10000000);
					OldVelocity[axisIdx]:= ExtVelocity[axisIdx];
					ExtDirection := SEL(TableOffsetPos[axisIdx] >= OldPosition[axisIdx], -1, 1);

					MC_ExtSetPointGenFeed(
						Position := TableOffsetPos[axisIdx],
						Velocity := ExtVelocity[axisIdx],
						Acceleration := ExtAcceleration,
						Direction := ExtDirection,
						Axis := Axis[axisIdx].Axis);
				END_IF
			END_FOR


			IF IsAutoRun THEN
				CurrentTableOffset := CurrentTableOffset + SubSpeed/100;
			ELSE
				CurrentTableOffset := CurrentTableOffset + Override/100;
			END_IF
			
			IF CurrentTableOffset >= 1 THEN
				CurrentTableOffset := CurrentTableOffset - 1;
				CurrentTableIdx := CurrentTableIdx + 1;
			END_IF

			IF CurrentTableIdx = SubProgramConfig[RunSubNo].TotalTableSize THEN
				SubRunAloneState := S_Complete;
				SubRunAloneFirstTime := TRUE;
				SubRunning := FALSE;
				FOR axisIdx:=1 TO No DO
					Axis[axisIdx].DisableSetPointGenerator.Execute := TRUE;
				END_FOR			
			END_IF


	END_CASE

END_IF

ACTION EnableExtSetPoint:


FOR axisIdx := 1 TO No DO
	IF AxisIsOn[axisIdx] THEN
		Axis[axisIdx].EnableSetPointGenerator
		(
			Execute := TRUE,
			Position := Axis[axisIdx].ActPos,
			PositionType := POSITIONTYPE_ABSOLUTE,
			Axis :=  Axis[axisIdx].Axis
		);
	END_IF
END_FOR
SubRunAloneState := S_WaitExtSetPoint;
END_ACTION

ACTION FillSubIOTable:
IF AirTableBuf.OK THEN
    FOR airIdx := 1 TO AirNo DO
        FOR Idx := 0 TO 1999  DO
			SubProgramTable[RunSubNo].airTable[airIdx, idx + SendOffset] := AirTableBuf.Table[airIdx, idx];
		END_FOR
	END_FOR
	SendOffset := SendOffset + 2000;
	AirTableBuf.OK := FALSE;
	IF SendOffset >= SubProgramConfig[RunSubNo].TotalTableSize THEN
		SendOffset := 0;
        SubRunAloneState := S_EnableExtSetPoint;
	END_IF
END_IF
IsGetTableBuf := AirTableBuf.OK;
END_ACTION

ACTION FillSubTable:
IF AxisTableBuf.OK THEN
	FOR axisIdx := 1 TO No DO
		FOR Idx := 0 TO 1999  DO
			SubProgramTable[RunSubNo].AxisTable[axisIdx, idx + SendOffset] := AxisTableBuf.Table[axisIdx, idx];
		END_FOR
	END_FOR
	SendOffset := SendOffset + 2000;
	AxisTableBuf.OK := FALSE;
	IF SendOffset >= SubProgramConfig[RunSubNo].TotalTableSize THEN
		SendOffset := 0;
        SubRunAloneState := S_FillSubIOTable;;
	END_IF
END_IF
IsGetTableBuf := AxisTableBuf.OK;
END_ACTION

ACTION Initial:

FOR axisIdx:=1 TO No DO
	(*Set的最後一個點非0的時候沒清會爆衝*)
	Axis[axisIdx].Axis.PlcToNc.ExtSetPos := Axis[axisIdx].ActPos;
	Axis[axisIdx].EnableSetPointGenerator.Execute := FALSE;
	TableOffsetPos[axisIdx] := Axis[axisIdx].ActPos;
	OldPosition[axisIdx] := Axis[axisIdx].ActPos;
	OldVelocity[axisIdx] := 0;
	IsExtSetPointDone[axisIdx]:=FALSE;
END_FOR

AxisTableBuf.OK		:= FALSE;

SubRunAloneFirstTime:= FALSE;
Idx0FirstTime		:= TRUE;
SubRunAloneState	:= S_FillSubTable;

(*Send Table*)
SendOffset			:= 0;

(*Index*)
CurrentTableIdx		:= 0;
CurrentTableOffset	:= 0;
END_ACTION

ACTION SubAirFunc:
(*----------------SubAir----------------1,2,7,8是探針汽缸*)
(*非測試編輯時跑表*)
IF NOT (Inputstate.VRSwitch = FALSE) THEN
	FOR airIdx := 1 TO AirNo DO
		IF  airIdx <> 1 
		AND airIdx <> 2 
		AND airIdx <> 7 
		AND airIdx <> 8
		THEN
			AirIsOpen[airIdx] := SubProgramTable[RunSubNo].AirTable[airIdx, CurrentTableIdx];
		END_IF
	END_FOR
END_IF
END_ACTION

ACTION WaitExtSetPoint:

IsSetPointComplete := TRUE;
FOR axisIdx := 1 TO No DO
	IF AxisIsOn[axisIdx] THEN
		IF Axis[axisIdx].EnableSetPointGenerator.Done THEN
			Axis[axisIdx].EnableSetPointGenerator.Execute := FALSE;
			IsExtSetPointDone[axisIdx] := TRUE;
		END_IF
		IsSetPointComplete := IsSetPointComplete AND IsExtSetPointDone[axisIdx];
	END_IF
END_FOR
IF IsSetPointComplete THEN
	SubRunAloneState := S_Run;
END_IF
END_ACTION

END_PROGRAM

// ---- POUs/MoveToColPos.TcPOU
PROGRAM MoveToColPos
VAR

    MoveToPosState :(S_FillTable,  S_EnableExtSetPoint, S_WaitExtSetPoint, S_Run, S_Complete);
	Idx0FirstTime		:BOOL;
	idx					:INT ;
	axisIdx				:INT;
	TotalTimeByMs		:LREAL;
	Table				:ARRAY [1..No, 0..1999] OF LREAL;
	CurrentTableIdx		:DINT;
	CurrentTableOffset	:REAL;


	AxisNeedRun			:ARRAY [1..No] OF BOOL;
	IsExtSetPointDone	:ARRAY [1..No] OF BOOL;
	IsSetPointComplete 	:BOOL;
	TableOffsetPos		:ARRAY [1..No] OF  LREAL;
	OldPosition			:ARRAY [1..No] OF LREAL;
	ExtVelocity			:ARRAY [1..No] OF LREAL;
	OldVelocity			:ARRAY [1..No] OF LREAL;
	ExtAcceleration		:LREAL;
	ExtDirection		:DINT;

END_VAR


IF MoveToColPosRunning THEN

	IF MoveToPosFirstTime THEN
		(*初始化*)
				Initial();
	END_IF

	CASE MoveToPosState OF

		S_FillTable:
						FillTable();

		S_EnableExtSetPoint:
						EnableExtSetPoint();

		S_WaitExtSetPoint:
						WaitExtSetPoint();

		S_Run:

			(* 表一開始 初始*)
			IF CurrentTableIdx = 0 AND Idx0FirstTime THEN
				Idx0FirstTime 		:= FALSE;
				OldPosition[axisIdx] 	:= 0;
				OldVelocity[axisIdx] 	:= 0;
			END_IF



			(*副程式*)

			(* 設定ExtPosition *)
			FOR axisIdx := 1 TO No DO
				IF AxisNeedRun[axisIdx] THEN
					(* 超過這條最後idx *)
					IF (CurrentTableIdx + CurrentTableOffset) > (TotalTimeByMs - 1) THEN
						TableOffsetPos[axisIdx]:= Table[axisIdx, CurrentTableIdx];
					ELSE
					(* idx在此表內 *)
						TableOffsetPos[axisIdx]:= Table[axisIdx, CurrentTableIdx] + ( Table[axisIdx, CurrentTableIdx + 1] - Table[axisIdx, CurrentTableIdx] ) * CurrentTableOffset;
					END_IF
				END_IF
			END_FOR

			FOR axisIdx := 1 TO No DO
				IF AxisNeedRun[axisIdx] THEN
					ExtVelocity[axisIdx]:= (TableOffsetPos[axisIdx] - OldPosition[axisIdx]) / (UDINT_TO_LREAL(_TaskInfo[1].CycleTime) / 10000000);
					OldPosition[axisIdx]:= TableOffsetPos[axisIdx];
					ExtAcceleration :=  (ExtVelocity[axisIdx] - OldVelocity[axisIdx]) / (UDINT_TO_LREAL(_TaskInfo[1].CycleTime) / 10000000);
					OldVelocity[axisIdx]:= ExtVelocity[axisIdx];
					ExtDirection := SEL(TableOffsetPos[axisIdx] >= OldPosition[axisIdx], -1, 1);

					MC_ExtSetPointGenFeed(
						Position := TableOffsetPos[axisIdx],
						Velocity := ExtVelocity[axisIdx],
						Acceleration := ExtAcceleration,
						Direction := ExtDirection,
						Axis := Axis[axisIdx].Axis);
				END_IF
			END_FOR

			CurrentTableOffset := CurrentTableOffset + Override/100;
			
			IF CurrentTableOffset >= 1 THEN
				CurrentTableOffset := CurrentTableOffset - 1;
				CurrentTableIdx := CurrentTableIdx + 1;
			END_IF

			IF CurrentTableIdx = TotalTimeByMs THEN
				MoveToPosState := S_Complete;
				MoveToPosFirstTime := TRUE;
				MoveToColPosRunning := FALSE;
				FOR axisIdx:=1 TO No DO
					Axis[axisIdx].DisableSetPointGenerator.Execute := TRUE;
				END_FOR			
			END_IF


	END_CASE

END_IF

ACTION EnableExtSetPoint:


FOR axisIdx := 1 TO No DO
	IF AxisNeedRun[axisIdx] THEN
		Axis[axisIdx].EnableSetPointGenerator
		(
			Execute := TRUE,
			Position := Axis[axisIdx].ActPos,
			PositionType := POSITIONTYPE_ABSOLUTE,
			Axis :=  Axis[axisIdx].Axis
		);
	END_IF
END_FOR
MoveToPosState := S_WaitExtSetPoint;
END_ACTION

ACTION FillTable:
IF AxisTableBuf.OK THEN
	FOR axisIdx := 1 TO No DO
		FOR Idx := 0 TO 1999  DO
			Table[axisIdx, idx] := AxisTableBuf.Table[axisIdx, idx];
		END_FOR
	END_FOR
	AxisTableBuf.OK := FALSE;
    MoveToPosState := S_EnableExtSetPoint;
END_IF
IsGetTableBuf := AxisTableBuf.OK;
END_ACTION

ACTION Initial:

FOR axisIdx:=1 TO No DO
	(*Set的最後一個點非0的時候沒清會爆衝*)
	Axis[axisIdx].Axis.PlcToNc.ExtSetPos := Axis[axisIdx].ActPos;
	Axis[axisIdx].EnableSetPointGenerator.Execute := FALSE;
	TableOffsetPos[axisIdx] := Axis[axisIdx].ActPos;
	OldPosition[axisIdx] := Axis[axisIdx].ActPos;
	OldVelocity[axisIdx] := 0;
	IsExtSetPointDone[axisIdx]:=FALSE;
END_FOR

AxisTableBuf.OK		:= FALSE;

MoveToPosFirstTime  := FALSE;
Idx0FirstTime		:= TRUE;
MoveToPosState		:= S_FillTable;

(*Index*)
CurrentTableIdx		:= 0;
CurrentTableOffset	:= 0;
END_ACTION

ACTION WaitExtSetPoint:

IsSetPointComplete := TRUE;
FOR axisIdx := 1 TO No DO
	IF AxisNeedRun[axisIdx] THEN
		IF Axis[axisIdx].EnableSetPointGenerator.Done THEN
			Axis[axisIdx].EnableSetPointGenerator.Execute := FALSE;
			IsExtSetPointDone[axisIdx] := TRUE;
		END_IF
		IsSetPointComplete := IsSetPointComplete AND IsExtSetPointDone[axisIdx];
	END_IF
END_FOR
IF IsSetPointComplete THEN
	MoveToPosState := S_Run;
END_IF
END_ACTION

END_PROGRAM

// ---- POUs/ManMove.TcPOU
PROGRAM ManMove
VAR
	ManMovState		: ARRAY[1..No] OF INT:=[No(MANMOVEENUM.S_MANINITIAL)];
	Stop			: BOOL;
	MPGIsSet		: BOOL:=FALSE;
	JogBoxIsSet		: BOOL;
	MinPosition		: ARRAY[1..No] OF LREAL;
	MaxPosition		: ARRAY[1..No] OF LREAL;
	FirstTime		: BOOL:= TRUE;
	idx				: INT;
	IsMpgMove		: BOOL:=FALSE;
	FeederCount		: INT:=0;
	AxisPos 			: ARRAY[1..No] OF REAL:=[No(0)];
	AxisLPos 		: ARRAY[1..No] OF REAL:=[No(0)];
	AxisPosByDist	: ARRAY[1..No] OF REAL:=[No(0)];
	UnitPos			: ARRAY[1..No] OF REAL:=[No(0)];
	RelativeMOVE	: RelativeMOVE;
	RelativeMOVE2	: RelativeMOVE2;
	ManMovCal		: ManMovCal;
	ReadActualPosition: MC_ReadActualPosition;
	RM1Busy		: ARRAY[1..No] OF BOOL:=[No(FALSE)];
	RM2Busy		: ARRAY[1..No] OF BOOL:=[No(TRUE)];

	Pos				: ARRAY[1..No] OF REAL:=[No(0)];
	Dist				: ARRAY[1..No] OF REAL:=[No(0)];
	Vel				: ARRAY[1..No] OF REAL:=[No(0)];
	Acc				: ARRAY[1..No] OF REAL:=[No(0)];
	Jerk 			: ARRAY[1..No] OF REAL:=[No(0)];

	AddFeederDist	: REAL;
	AddFeederV		: REAL;
	AddFeederAcc	: REAL;
	AddFeederJerk	: REAL;

	mem			: ARRAY[1..1000] OF REAL;
	memIdx			: INT := 1;
	count			: INT:=1;
	FirstPos			: ARRAY[1..No] OF LREAL;
END_VAR


IF State = ENUMSTATE.S_MANMOV OR State = ENUMSTATE.S_TROSHO_MANMOV THEN
	IF FirstTime THEN
		FirstTime := FALSE;
		(*給定手動起始位置*)
		FOR idx := 1 TO No DO
			Pos[idx] := FirstPos[idx];
		END_FOR
		(*初始化電子凸輪狀態Decouple*)
		FOR idx:=1 TO No DO
			Cam[idx].CamOut(Execute := TRUE, Slave:=Axis[idx].Axis);
		END_FOR
	END_IF
	(*------------------------手輪---------------------------*)
	IF MPGIsSet THEN
		IF AxisIsOn[CurManMovAxis] THEN
			IF Mpg_PositiveMove = TRUE THEN
				IsMpgMove :=TRUE;
				AxisManMove[CurManMovAxis].Execute := TRUE;
				IF AxisManMove[CurManMovAxis].DistByUnit < 0 THEN
					AxisManMove[CurManMovAxis].DistByUnit := -AxisManMove[CurManMovAxis].DistByUnit;
				END_IF
			ELSIF Mpg_NegativeMove = TRUE THEN
				IsMpgMove :=TRUE;
				AxisManMove[CurManMovAxis].Execute := TRUE;
				IF AxisManMove[CurManMovAxis].DistByUnit > 0 THEN
					AxisManMove[CurManMovAxis].DistByUnit := -AxisManMove[CurManMovAxis].DistByUnit;
				END_IF
			ELSIF Inputstate.Mpg_PositiveBtn = TRUE THEN
				IsMpgMove :=TRUE;
				AxisManMove[CurManMovAxis].Execute := TRUE;
				IF AxisManMove[CurManMovAxis].DistByUnit < 0 THEN
					AxisManMove[CurManMovAxis].DistByUnit := -AxisManMove[CurManMovAxis].DistByUnit;
				END_IF	
			ELSIF Inputstate.Mpg_NegativeBtn = TRUE THEN
				IsMpgMove :=TRUE;
				AxisManMove[CurManMovAxis].Execute := TRUE;
				IF AxisManMove[CurManMovAxis].DistByUnit > 0 THEN
					AxisManMove[CurManMovAxis].DistByUnit := -AxisManMove[CurManMovAxis].DistByUnit;
				END_IF
			ELSIF IsMpgMove = TRUE THEN
				IsMpgMove :=FALSE;
				AxisManMove[CurManMovAxis].Execute := FALSE;
			END_IF
		END_IF
	(*------------------------吋動盒-------------------------*)
	ELSIF JogBoxIsSet THEN
		IF Inputstate.plusY THEN
			AxisManMove[FeederNo].Execute := TRUE;
			IF AxisManMove[FeederNo].DistByUnit < 0 THEN
				AxisManMove[FeederNo].DistByUnit := -AxisManMove[FeederNo].DistByUnit;
			END_IF
		ELSIF Inputstate.negY THEN
			AxisManMove[FeederNo].Execute := TRUE;
			IF AxisManMove[FeederNo].DistByUnit > 0 THEN
				AxisManMove[FeederNo].DistByUnit := -AxisManMove[FeederNo].DistByUnit;
			END_IF
		ELSIF Inputstate.plusA THEN
			AxisManMove[RotateWNo].Execute := TRUE;
			IF AxisManMove[RotateWNo].DistByUnit < 0 THEN
				AxisManMove[RotateWNo].DistByUnit := -AxisManMove[RotateWNo].DistByUnit;
			END_IF
			AxisManMove[FeederNo].Execute := TRUE;
			IF AxisManMove[FeederNo].DistByUnit < 0 THEN
				AxisManMove[FeederNo].DistByUnit := -AxisManMove[FeederNo].DistByUnit;
			END_IF
		ELSIF Inputstate.negA THEN
			AxisManMove[RotateWNo].Execute := TRUE;
			IF AxisManMove[RotateWNo].DistByUnit > 0 THEN
				AxisManMove[RotateWNo].DistByUnit := -AxisManMove[RotateWNo].DistByUnit;
			END_IF
			AxisManMove[FeederNo].Execute := TRUE;
			IF AxisManMove[FeederNo].DistByUnit > 0 THEN
				AxisManMove[FeederNo].DistByUnit := -AxisManMove[FeederNo].DistByUnit;
			END_IF
		ELSE
			AxisManMove[RotateWNo].Execute := FALSE;
			AxisManMove[FeederNo].Execute := FALSE;
			JogBoxIsSet := FALSE;
		END_IF
	END_IF


	IF Stop THEN
		Stop := FALSE;
		FOR idx:= 1 TO No DO
			AxisManMove[idx].Execute := FALSE;
		END_FOR
	END_IF

	FOR idx:= 1 TO No DO
		IF AxisManMove[idx].DistByUnit <>0 THEN
			ReadActualPosition(Enable:=TRUE, Axis:=Axis[idx].Axis);
			AxisPos[idx] := ReadActualPosition.Position;
			AxisPosByDist[Idx]   := AxisPosByDist[Idx] +  AxisPos[Idx] - AxisLPos[Idx];
			AxisLPos[Idx]     	    := AxisPos[Idx];

			CASE ManMovState[idx] OF
				MANMOVEENUM.S_MANINITIAL:
					IF AxisManMove[idx].Execute THEN
						(*Override := 100;(*手動調回100%*)*)
						(*第一個相對運動判斷目前是否為靜止*)
							AxisPosByDist[idx]      := 0;
							ManMovCal(
								Axis 	:= idx,
								Pos		:= Pos[idx],
								MinPos	:= MinPosition[idx],
								MaxPos  := MaxPosition[idx],
								NPos	=>Pos[idx],
								Dist		=>Dist[idx],
								Vel     	=>Vel[idx],
								Acc     	=>Acc[idx],
								Jerk   	=>Jerk[idx]
							);

							IF Dist[idx] <> 0 THEN
								RelativeMOVE(
									MoveAxisIdx		:= idx,
									MoveDistance	:= Dist[idx],
									MoveVelocity		:= Vel[idx],
									MoveAcceleration:= Acc[idx]*0.1,
									MoveDeceleration:= Acc[idx]*2,
									MoveJerk	   	 := Jerk[idx]
								);
								(*翻線捕線*)
								IF idx = RotateWNo THEN
									AddFeederDist  :=  Dist[idx] * RWAddFeederRatio;
									AddFeederV       :=  ABS( Vel[idx] * RWAddFeederRatio );
									AddFeederAcc  :=  ABS(AddFeederV/AxisManMove[idx].AccTime);
									AddFeederJerk :=  AddFeederAcc/0.0001;
									RelativeMOVE(
										MoveAxisIdx		:= FeederNo,
										MoveDistance	:= AddFeederDist,
										MoveVelocity		:= AddFeederV ,
										MoveAcceleration := AddFeederAcc*0.1,
										MoveDeceleration := AddFeederAcc*2,
										MoveJerk	   	 := AddFeederJerk,
									);
								END_IF
								ManMovState[idx] := MANMOVEENUM.S_MANMOVE;
							END_IF
					END_IF

				MANMOVEENUM.S_MANMOVE:
					IF AxisManMove[idx].Execute THEN

						(*起始動作送完接著後續連續運動*)
						IF ABS(AxisPosByDist[Idx])  >= ABS(Dist[idx]* 9.0/10.0) THEN

							 IF ABS(AxisPosByDist[Idx])  >= ABS(Dist[idx]) THEN
								IF AxisManMove[CurManMovAxis].DistByUnit > 0 THEN
									AxisPosByDist[Idx] := AxisPosByDist[Idx] - Dist[idx];
								ELSE
									AxisPosByDist[Idx] := AxisPosByDist[Idx] + Dist[idx];
								END_IF
							END_IF


							IF  (Axis[idx].fbMC_MoveRelative[1].Busy=FALSE) AND Axis[idx].fbMC_MoveRelative[2].Busy THEN

								AxisPosByDist[idx]      := 0;

								ManMovCal(
									Axis 	:= idx,
									Pos		:= Pos[idx],
									MinPos	:= MinPosition[idx],
									MaxPos  := MaxPosition[idx],
									NPos	=>Pos[idx],
									Dist		=>Dist[idx],
									Vel     	=>Vel[idx],
									Acc     	=>Acc[idx],
									Jerk    	=>Jerk[idx]
								);
								IF Dist[idx] <> 0 THEN
									RelativeMOVE(
										MoveAxisIdx		:= idx,
										MoveDistance	:= Dist[idx],
										MoveVelocity		:= Vel[idx],
										MoveAcceleration:= Acc[idx]*0.1,
										MoveDeceleration:= Acc[idx]*2,
										MoveJerk	 	:= Jerk[idx]
										);
									(*翻線捕線*)
									IF idx = RotateWNo THEN
										AddFeederDist  :=  Dist[idx] * RWAddFeederRatio;
										AddFeederV       :=  ABS( Vel[idx] * RWAddFeederRatio);
										AddFeederAcc  :=  ABS(AddFeederV/AxisManMove[idx].AccTime);
										AddFeederJerk :=  AddFeederAcc/0.0001;
										RelativeMOVE(
											MoveAxisIdx		:= FeederNo,
											MoveDistance	:= AddFeederDist,
											MoveVelocity		:= AddFeederV ,
											MoveAcceleration := AddFeederAcc*0.1,
											MoveDeceleration := AddFeederAcc*2,
											MoveJerk	   	 := AddFeederJerk,
										);
									END_IF
								END_IF
							ELSIF Axis[idx].fbMC_MoveRelative[1].Busy AND (Axis[idx].fbMC_MoveRelative[2].Busy=FALSE) THEN

								AxisPosByDist[idx]      := 0;

								ManMovCal(
									Axis 	:= idx,
									Pos		:= Pos[idx],
									MinPos	:= MinPosition[idx],
									MaxPos  := MaxPosition[idx],
									NPos	=>Pos[idx],
									Dist		=>Dist[idx],
									Vel     	=>Vel[idx],
									Acc     	=>Acc[idx],
									Jerk   	 =>Jerk[idx]
								);
								IF Dist[idx] <> 0 THEN
									RelativeMOVE2(
										MoveAxisIdx		:= idx,
										MoveDistance	:= Dist[idx],
										MoveVelocity		:= Vel[idx],
										MoveAcceleration:= Acc[idx]*0.1,
										MoveDeceleration:= Acc[idx]*2,
										MoveJerk	  	:= Jerk[idx]
									);
									(*翻線捕線*)
									IF idx = RotateWNo THEN
										AddFeederDist  :=  Dist[idx] * RWAddFeederRatio;
										AddFeederV       := ABS( Vel[idx] * RWAddFeederRatio);
										AddFeederAcc  :=  ABS(AddFeederV/AxisManMove[idx].AccTime);
										AddFeederJerk :=  AddFeederAcc/0.0001;
										RelativeMOVE2(
											MoveAxisIdx		:= FeederNo,
											MoveDistance	:= AddFeederDist,
											MoveVelocity		:= AddFeederV ,
											MoveAcceleration := AddFeederAcc*0.1,
											MoveDeceleration := AddFeederAcc*2,
											MoveJerk	   	 := AddFeederJerk,
										);
									END_IF
								END_IF

							END_IF
						END_IF
					ELSE
						ManMovState[idx] := MANMOVEENUM.S_MOVESTOP;
					END_IF

				MANMOVEENUM.S_MOVESTOP:
					IF (Axis[idx].fbMC_MoveRelative[1].Busy=FALSE) AND (Axis[idx].fbMC_MoveRelative[2].Busy=FALSE) THEN
						ManMovState[idx] := MANMOVEENUM.S_MANINITIAL;
					END_IF
			END_CASE
		END_IF
	END_FOR





(*-----------------------若不是手動----------------------*)
ELSE
	FirstTime := TRUE;
END_IF

END_PROGRAM

// ---- POUs/FB/ManMovCal.TcPOU
FUNCTION_BLOCK ManMovCal
VAR_INPUT
	Axis			: INT;
	Pos			: LREAL;
	MinPos		: LREAL;
	MaxPos   	: LREAL;
END_VAR
VAR_OUTPUT
	NPos	: LREAL;
	Dist		: LREAL;
	Vel		: LREAL;
	Acc		: LREAL;
	Jerk		: LREAL;
END_VAR
VAR
	StartPos		: DINT;
	EndPos		: DINT;
END_VAR

StartPos := LREAL_TO_DINT(Pos * AxisManMove[Axis].UnitRatio);(*單位轉換有四捨五入功能 超過DINT大小仍可運作正常*)
NPos := Pos  +  AxisManMove[Axis].DistByUnit ;

IF NPos < MinPos THEN
	IF NPos <= Pos THEN (* 反向移動 *)
		IF Pos < MinPos THEN (* 目前已經小於最小值位置 不動*)
			NPos := Pos;
		ELSE (* 目前位置還沒到達最大值 *)
			NPos := MinPos;
		END_IF
	END_IF
ELSIF NPos > MaxPos THEN
	IF NPos >= Pos THEN (* 正向移動 *)
		IF Pos > MaxPos THEN (* 目前已經大於最大值位置 不動*)
			NPos := Pos;
		ELSE (* 目前位置還沒到達最大值 *)
			NPos := MaxPos;
		END_IF
	END_IF
END_IF

EndPos  := LREAL_TO_DINT((NPos) * AxisManMove[Axis].UnitRatio);

Dist := DINT_TO_LREAL(EndPos - StartPos);

Vel := ABS( Dist  / (AxisManMove[Axis].MoveTime - AxisManMove[Axis].AccTime) ) ;

(* S-Curve
Acc := 2*Vel /( (1 + (1 - (0.01*AxisManMove[Axis].JerkP))) * AxisManMove[Axis].AccTime );
Jerk:= (200 / AxisManMove[Axis].JerkP) * (Acc  / AxisManMove[Axis].AccTime);
*)

(*T-Curve*)
Acc := ABS(Vel/AxisManMove[Axis].AccTime);
Jerk:= Acc/0.0001;

END_FUNCTION_BLOCK

// ---- POUs/HomeByTouchProbe.TcPOU
PROGRAM HomeByTouchProbe
VAR
	ENUMHOMINGSTATE  : (S_STARTHOMING, S_RESET, S_DELAYFORSTOP, S_MOVETONEWZERO, S_DELAYFORSTOP2, S_SETPOSITION, S_HOMINGCOMPLETE);
	HomingST			  : ARRAY [1..No] OF ST_TouchProbeHomeByUI;
	HomingStart			  : ARRAY [1..No] OF BOOL;
	HomingState			  : ARRAY [1..No] OF INT;
	idx 				           : INT;
	ActPos   				  : LREAL;
	MoveDis			 	  : LREAL;
	Trig1				  : ARRAY [1..No] OF R_TRIG;
	Trig2				  : ARRAY [1..No] OF R_TRIG;
	Trig3				  : ARRAY [1..No] OF R_TRIG;
	Timer			 	  : ARRAY [1..No] OF TON;
	Timer2			 	  : ARRAY [1..No] OF TON;
	FB_TouchProbe		  : FB_TouchProbe;
	RelativeMOVE 	 	  : RelativeMOVE;
	GetActPos			  : MC_ReadActualPosition;
	posset				  : LREAL;
	PosNear				  : FB_PosNear;
	PosIsNear			  : BOOL:=FALSE;
	CloseAir				  : FB_CloseAir;
END_VAR

IF State = ENUMSTATE.S_ZRT THEN
	IF ZRTFirstTime = TRUE THEN
		(*Override		:= 100;*)
		ZRTFirstTime := FALSE;
		PosIsNear	 := FALSE;
		IF IsZrtGrpSelect = FALSE THEN
			(*非選軸回原點時, 汽缸初始化*)
						CloseAir();
	    END_IF
		(*初始化電子凸輪狀態Decouple*)
		FOR idx:=1 TO No DO
			Cam[idx].CamOut(Execute := TRUE, Slave:=Axis[idx].Axis);
		END_FOR
		FOR idx := 1 TO No DO
			HomingState[idx] := S_STARTHOMING;
			AxisTouchProbe[idx].Execute := FALSE;
			Trig1[idx](CLK:= FALSE);
			Trig2[idx](CLK:= FALSE);
			Trig3[idx](CLK:= FALSE);
		END_FOR
	END_IF

	FOR idx:=1 TO No DO
		IF HomingST[idx].Execute = TRUE THEN
			HomingStart[idx] := TRUE;
		END_IF

		IF HomingStart[idx] = TRUE THEN

			CASE HomingState[idx] OF
				S_STARTHOMING:(*開始回SENSOR原點*)
					FB_TouchProbe(AxisIdx:=idx);(*開始抓SENSOR原點位置*)
					AxisValue[idx].Jog_JogForward := TRUE;(*正向往原點方向移動*)
					AxisValue[idx].Jog_Mode		     := MC_JOGMODE_CONTINOUS;
					AxisValue[idx].Jog_Velocity		     := HomingST[idx].ZRTSpeed;(*歸零速度要使用變速*)
					HomingState[idx] := S_RESET;
				S_RESET:(*到達SENSOR原點急停*)
					IF AxisTouchProbe[idx].RecordPosition <> 0 THEN(*抓到原點表示走到*)
						Trig1[idx](CLK:= TRUE);
						Axis[idx].fbMC_Reset(
							Execute:=Trig1[idx].Q,
							Axis:=Axis[idx].Axis
						);
						AxisValue[idx].Jog_JogForward:= FALSE;
						IF Axis[idx].fbMC_Reset.Done = TRUE THEN
							Trig1[idx](CLK:=FALSE);
							HomingState[idx] := S_DELAYFORSTOP;
						END_IF
					END_IF
				S_DELAYFORSTOP:(*等待軸確實停止*)
					PosNear(AxisIdx:=idx, Offset:=5, IsNear=>PosIsNear);
					IF PosIsNear = TRUE THEN
						PosIsNear := FALSE;
						HomingState[idx] := S_MOVETONEWZERO;
					END_IF
				S_MOVETONEWZERO:(*移動到新設原點*)
					Trig2[idx](CLK:= TRUE);
					IF Trig2[idx].Q = TRUE THEN
						GetActPos(Enable:=TRUE, Axis:=Axis[idx].Axis, Position=>ActPos);
						MoveDis := AxisTouchProbe[idx].RecordPosition -  ActPos + HomingST[idx].ZRTSet ;(*要再加上新設原點位置*)
						RelativeMOVE(
							MoveAxisIdx		:= idx,
							MoveDistance	:= MoveDis,
							MoveVelocity		:= HomingST[idx].ZRTSpeed
						);
					END_IF
					IF Axis[idx].fbMC_MoveRelative[1].Done = TRUE THEN
						Trig2[idx](CLK:=FALSE);
						HomingState[idx] := S_DELAYFORSTOP2;
					END_IF
				S_DELAYFORSTOP2:(*等待移動確實停止*)
					PosNear(AxisIdx:=idx, Offset:=2, IsNear=>PosIsNear);
					IF PosIsNear = TRUE THEN
						PosIsNear := FALSE;
						HomingState[idx] := S_SETPOSITION;
					END_IF
				S_SETPOSITION:(*將新設原點位置設成0*)
					GetActPos(Enable:=TRUE, Axis:=Axis[idx].Axis, Position=>ActPos);
					Trig3[idx](CLK:=TRUE);
					IF Trig3[idx].Q = TRUE THEN
						Axis[idx].fbMC_SetPosition(
							Execute	:= Trig3[idx].Q,
							Position	:= 0,
							Axis		:= Axis[idx].Axis
						);
					END_IF
					IF Axis[idx].fbMC_SetPosition.Done = TRUE THEN
						Trig3[idx](CLK:=FALSE);
						HomingState[idx] := S_HOMINGCOMPLETE;
					END_IF
				S_HOMINGCOMPLETE:(*歸零完成*)
					(*------------------------初始化-------------------------*)
					HomingStart[idx] 	:= FALSE;
					(*-----------------------------------------------------------*)
			END_CASE;
	
		END_IF
	END_FOR
END_IF

END_PROGRAM

// ---- POUs/FB/FB_TouchProbe.TcPOU
FUNCTION_BLOCK FB_TouchProbe
VAR_INPUT
	AxisIdx	:INT;
END_VAR
VAR_OUTPUT
END_VAR
VAR
END_VAR

AxisTouchProbe[AxisIdx].Execute := TRUE;

END_FUNCTION_BLOCK

// ---- POUs/FB/FB_PosNear.TcPOU
FUNCTION_BLOCK FB_PosNear
VAR_INPUT
	AxisIdx		: INT;
	Offset		: LREAL;
END_VAR
VAR_OUTPUT
	IsNear		: BOOL:=FALSE;
END_VAR
VAR
	ActPos		: LREAL;
	SetPos		: LREAL;
	ActMSet		: LREAL;
	OffsetByCount: LREAL;
	Scaling		: LREAL:=1;
END_VAR

IsNear			 := FALSE;
ActPos			 := Axis[AxisIdx].Axis.NcToPlc.ActPos;
SetPos			 := Axis[AxisIdx].Axis.NcToPlc.SetPos;
ActMSet			 := ABS(ActPos - SetPos);
OffsetByCount	 := Offset*Scaling;
IF  ActMSet <= OffsetByCount THEN
	IsNear	:= TRUE;
END_IF

END_FUNCTION_BLOCK

// ---- POUs/SetPosByUI.TcPOU
PROGRAM SetPosByUI
VAR
	SetPosST	: ST_SetPosByUI;
END_VAR

Axis[SetPosST.Axis].fbMC_SetPosition(
	Execute	:= SetPosST.Execute,
	Position	:= SetPosST.Position,
	Axis		:= Axis[SetPosST.Axis].Axis
);
SetPosST.Execute := FALSE;

END_PROGRAM

// ---- POUs/MCRelativeMove.TcPOU
PROGRAM MCRelativeMove
VAR
	RelativeMOVE	: ARRAY [1..No] OF MC_MoveRelative;
	Input			: ARRAY [1..No] OF ST_MCRelativeInput;
	Output			: ARRAY [1..No] OF ST_MCRelativeOutput;
	Trig				: ARRAY [1..No] OF R_TRIG;
	idx				: INT;
END_VAR

FOR idx:=1 TO No DO
	IF Input[idx].Execute = TRUE THEN
		Trig[idx](CLK := TRUE);
	ELSE
		Trig[idx](CLK := FALSE);
	END_IF
	RelativeMOVE[idx](
		Execute  			:= Trig[idx].Q,
		Distance			:= Input[idx].Distance,
		Velocity  			:= Input[idx].Velocity,
		Acceleration  		:= Input[idx].Acceleration,
		Deceleration 		:= Input[idx].Deceleration,
		Jerk				:= Input[idx].Jerk,
		Axis				:= Axis[idx].Axis,

		Done 			=> Output[idx].Done,
		Busy 			=> Output[idx].Busy,
		Active 			=> Output[idx].Active,
		CommandAborted => Output[idx].CommandAborted,
		Error 			=> Output[idx].Error,
		ErrorID 			=> Output[idx].ErrorID
	);
END_FOR

END_PROGRAM

// ---- POUs/AlertLight.TcPOU
PROGRAM AlertLight
VAR
	Light		: ST_AlertLight;
END_VAR

IF state = ENUMSTATE.S_AUTO THEN
	IF TouchMissStop OR SpeedDownTo0 THEN
		Light.Red := TRUE;
	ELSE
		Light.Green := TRUE;
	END_IF
ELSIF state = ENUMSTATE.S_ERROR OR state =  ENUMSTATE.S_TROUBLESHOOT OR state = ENUMSTATE.S_TROSHO_MANMOV OR TouchMissStop OR SpeedDownTo0 THEN
	Light.Red := TRUE;
ELSE
	Light.Orange := TRUE;
END_IF

IF MachineSubType = MachineSubTypeEnum.CE THEN

	IF Light.Orange THEN
		LightOGR[1] := TRUE;
		LightOGR[2] := FALSE;
		LightOGR[3] := FALSE;

	ELSIF Light.Green THEN
		LightOGR[1] := FALSE;
		LightOGR[2] := FALSE;
		LightOGR[3] := TRUE;
	
	ELSIF Light.Red THEN
		LightOGR[1] := FALSE;
		LightOGR[2] := TRUE;
		LightOGR[3] := FALSE;

	END_IF

ELSE

	IF Light.Orange THEN
		LightOGR[1] := FALSE;
		LightOGR[2] := FALSE;
		LightOGR[3] := FALSE;

	ELSIF Light.Green THEN
		LightOGR[1] := TRUE;
		LightOGR[2] := FALSE;
		LightOGR[3] := FALSE;
	
	ELSIF Light.Red THEN
		LightOGR[1] := FALSE;
		LightOGR[2] := TRUE;
		LightOGR[3] := FALSE;

	END_IF

END_IF

Light.Orange := FALSE;
Light.Green := FALSE;
Light.Red := FALSE;

END_PROGRAM

// ---- POUs/AxisStatusDataStore.TcPOU
PROGRAM AxisStatusDataStore
VAR
	idx				: INT:=1;
	count			: INT:=0;
END_VAR

FOR idx:=1 TO No DO
	RingBufferAxesPosBuf[idx].SetPos[count] := Axis[Idx].Axis.NcToPlc.SetPos;
	RingBufferAxesPosBuf[idx].ActPos[count] := Axis[Idx].Axis.NcToPlc.ActPos;
	RingBufferAxesVelBuf[idx].SetVel[count] := Axis[Idx].Axis.NcToPlc.SetVelo;
	RingBufferAxesVelBuf[idx].ActVel[count] := Axis[Idx].Axis.NcToPlc.ActVelo;
	RingBufferAxesTrqBuf[idx].Trq[count] := AxesTorque[Idx];
END_FOR

IF count = 999 THEN
	count := 0;
ELSE
	count := count + 1;
END_IF

END_PROGRAM

// ---- POUs/EncoderClear.TcPOU
PROGRAM EncoderClear
VAR
	Run		: BOOL:=FALSE;
	ClearAxis: ARRAY [1..No] OF BOOL;

	EnCLr	: FB_EncoderClear;
END_VAR

IF Run THEN
	EnCLr(ClearAxis := ClearAxis);
	IF EnClr.Busy = FALSE THEN
		Run := FALSE;
	END_IF
END_IF

END_PROGRAM

// ---- POUs/FB/FB_EncoderClear.TcPOU
FUNCTION_BLOCK FB_EncoderClear

VAR_INPUT
	ClearAxis	: ARRAY [1..No] OF BOOL;
END_VAR

VAR_OUTPUT
	Busy		: BOOL;
END_VAR

VAR
	exe			: ARRAY [1..No] OF BOOL;
	idx			: INT := 1;
	Value		: UINT := 16#10;
	Cmdstring	: STRING(16);
	deltaState	: UINT:=0;
	EnClrState	: UINT:=0;
	Timer		:TON;
	FirstTime	:BOOL:= TRUE;
	YASKAWAEnClr	: ARRAY [1..No] OF Y_AbsoluteEncoderReset;
END_VAR


IF MotorVendor = MotorVenderEnum.SANYO THEN
	Value := 16#10;
	FOR Idx := 1 TO No DO
		IF ClearAxis[idx] = TRUE THEN
			Axis[idx].fbADSWrite(
				NETID		:= AmsNetId,
				PORT		:= 501,
				IDXGRP		:= 16#F030,
				IDXOFFS	:= 16#B1 + (idx - 1)*16#D0, (*NC->Axis->Drive->Output->nCtrl1*)
				LEN			:= 1,
				SRCADDR 	:= ADR(Value),
				WRITE		:= TRUE,
				TMOUT		:=  t#0.5s,
			);
		END_IF
	END_FOR

	Busy := FALSE;
	FOR idx := 1 TO No DO
		IF ClearAxis[idx] = TRUE THEN
			IF  Axis[idx].fbADSWrite.BUSY THEN
				Busy := TRUE;
			END_IF
		END_IF
	END_FOR


ELSIF MotorVendor = MotorVenderEnum.YASKAWA THEN

	Busy := TRUE;

	FOR Idx := 1 TO No DO
		IF ClearAxis[idx] = TRUE THEN
			YASKAWAEnClr[idx](
				bExecute:= TRUE,
				sNetId:= DeviceNetId,
				nSlaveAddr:=  1009 + (Idx-1),
				bDone=> ,
				bBusy=> ,
				bError=> ,
				nErrorID=> );
		END_IF
	END_FOR


	Timer(IN:= TRUE,PT:= T#500ms );
	IF Timer.Q THEN
		Timer(IN:= FALSE);
		busy := FALSE;
	END_IF

ELSIF MotorVendor = MotorVenderEnum.DELTA THEN
(*可利用面版操作或是通訊寫入參數P2-71 為1 建立絕對型原點座標，當P2-71 被寫入1 時，
絕對系統座標會立刻進行重置。但因參數P2-71 寫入功能受到P2-08 保護，必須先寫入參數
P2-08 為271，才能順利寫入參數P2-71。因此，參數的輸入順序為P2-08 = 271，然後是
P2-71 = 1。請注意，此方法只適合PR 以外的模式使用。若是操作在PR 模式，請使用原點
復歸的程序建立絕對型原點座標。*)

	IF FirstTime THEN
		FirstTime := FALSE;
		FOR Idx := 1 TO No DO
			exe[idx] := TRUE;
		END_FOR
	END_IF
	Busy := TRUE;
	CASE deltaState OF
		0:
			FOR Idx := 1 TO No DO
				IF ClearAxis[idx] = TRUE THEN
					Value := 271;
					Axis[idx].fbSDOWrite(
						bExecute 	:= exe[idx],
						sNetId 		:= DeviceNetId,
						nSlaveAddr 	:= 1009 + (Idx-1),
						nIndex 		:= 16#2208,
						nSubIndex 	:= 0,
						pSrcBuf 		:= ADR(Value),
						cbBufLen 	:= SIZEOF(Value)
					);
					IF NOT Axis[idx].fbSDOWrite.bBusy THEN
						exe[idx] := FALSE;
					END_IF
				END_IF
			END_FOR
			Timer(IN:= TRUE,PT:= T#500ms );
			IF Timer.Q THEN
				Timer(IN:= FALSE);
				deltaState := 1;
				FOR Idx := 1 TO No DO
					exe[idx] := TRUE;
				END_FOR
			END_IF
		1:
			FOR Idx := 1 TO No DO
				IF ClearAxis[idx] = TRUE THEN
					Value := 1;
					Axis[idx].fbSDOWrite(
						bExecute 	:= exe[idx],
						sNetId 		:= DeviceNetId,
						nSlaveAddr 	:= 1009 + (Idx-1),
						nIndex 		:= 16#2247,
						nSubIndex 	:= 0,
						pSrcBuf 		:= ADR(Value),
						cbBufLen 	:= SIZEOF(Value)
					);
					IF NOT Axis[idx].fbSDOWrite.bBusy THEN
						exe[idx] := FALSE;
					END_IF
				END_IF
			END_FOR
			Timer(IN:= TRUE,PT:= T#500ms );
			IF Timer.Q THEN
				Timer(IN:= FALSE);
				deltaState := 4;
				FOR Idx := 1 TO No DO
					exe[idx] := TRUE;
				END_FOR
			END_IF
		4:
			Busy := FALSE;
	END_CASE
END_IF

END_FUNCTION_BLOCK

// ---- POUs/UPS.TcPOU
PROGRAM UPS
VAR
	fbGetUPSStatus	: FB_GetUPSStatus;(*Cx20x0*)

	Timer			: TON;
	PowerFailTrig	: R_TRIG;

	fb51x0UPS		: FB_S_UPS_CX51x0;			(* UPS-FB instance *)
	eUpsMode		: E_S_UPS_Mode	:= eSUPS_CheckPowerStatus; (* UPS mode (writing persistent data + shutdown) *)

	fbWritePersistentData	:FB_WritePersistentData;
END_VAR
VAR PERSISTENT
	powerFailCount1 	:UDINT;
	powerFailCount2 	:UDINT;
END_VAR


IF DeviceNetId <> '' THEN
	fbGetUPSStatus(bEnable := TRUE);

	IF NOT fbGetUPSStatus.bError THEN
		IF fbGetUPSStatus.stStatus.ePowerStatus = PowerOnBattery THEN
			PowerFailTrig(CLK:= TRUE);
			IF PowerFailTrig.Q THEN
				InPowerOffProcess := TRUE;
			END_IF
		ELSE
			IF PowerFailTrig.M AND InPowerOffProcess THEN
				InPowerOffProcess := FALSE;
			END_IF
			PowerFailTrig(CLK:= FALSE);
		END_IF
(*	ELSE
CX51xx
fb51x0UPS(eUpsMode := eUpsMode);
eGlobalSUpsState: Internal state of the function block as global copy of VAR_OUTPUT*)
(*
IF eGlobalSUpsState >= eSUPS_PowerFailure THEN
			Inputstate.PowerOff := TRUE;
		ELSE
			Inputstate.PowerOff := FALSE;
		END_IF
*)
	END_IF
END_IF

END_PROGRAM

// ---- POUs/CoEConfig.TcPOU
PROGRAM CoEConfig
VAR
END_VAR

;

END_PROGRAM

// ---- POUs/FB/FB_CheckInfoData.TcPOU
FUNCTION_BLOCK FB_CheckInfoData
VAR_INPUT
	Decimal		: INT;
END_VAR
VAR_OUTPUT
	IsError	    :BOOL;
END_VAR
VAR
	count		: INT;
	Hex0		: DWORD;
	Hex1		: DWORD;
	Hex2		: DWORD;
	Hex3		: DWORD;
END_VAR

count := 0;
Hex0:= 0; Hex1:= 0; Hex2:=0; Hex3:=0;
WHILE Decimal > 0 DO
	CASE count OF
		0:
			Hex0 := Decimal MOD 16;
		1:
			Hex1 := Decimal MOD 16;
		2:
			Hex2 := Decimal MOD 16;
		3:
			Hex3 := Decimal MOD 16;
	END_CASE;
	Decimal := Decimal / 16;
	count := count + 1;
END_WHILE

IF Hex0 <> 8 OR Hex1 <> 0 OR Hex2 <> 0 OR Hex3 <> 0 THEN
	IsError := TRUE;
END_IF

END_FUNCTION_BLOCK

// ---- POUs/FB/FB_GetExtPosition.TcPOU
FUNCTION_BLOCK FB_GetExtPosition
VAR_INPUT
	tableIdx		: DINT;
	tableOffset	: LREAL;
END_VAR
VAR_OUTPUT
END_VAR
VAR
END_VAR

;

END_FUNCTION_BLOCK

// ---- POUs/FB/MasterMove.TcPOU
FUNCTION_BLOCK MasterMove
VAR_INPUT
	MoveDistance		: LREAL;
	MoveVelocity			: LREAL;
	MoveAcceleration		: LREAL;
	MoveDeceleration		: LREAL;
	MoveJerk			: LREAL;
END_VAR
VAR_OUTPUT
END_VAR
VAR
END_VAR


Master.fbMC_MoveRelative[1](
	Execute  		:= TRUE,
	Distance		:= MoveDistance,
	Velocity  		:= MoveVelocity,
	Acceleration   := MoveAcceleration,
	Deceleration  := MoveDeceleration,
	Jerk			:= MoveJerk,
	BufferMode     := MC_BlendingHigh,
	Axis			:= Master.Axis
);

Master.fbMC_MoveRelative[1](
	Execute  		:= FALSE,
	Axis			:= Master.Axis
);

END_FUNCTION_BLOCK

// ---- POUs/FB/MasterMove2.TcPOU
FUNCTION_BLOCK MasterMove2
VAR_INPUT
	MoveDistance		: LREAL;
	MoveVelocity			: LREAL;
	MoveAcceleration		: LREAL;
	MoveDeceleration		: LREAL;
	MoveJerk			: LREAL;
END_VAR
VAR_OUTPUT
END_VAR
VAR
END_VAR


Master.fbMC_MoveRelative[2](
	Execute  		:= TRUE,
	Distance		:= MoveDistance,
	Velocity  		:= MoveVelocity,
	Acceleration   := MoveAcceleration,
	Deceleration  := MoveDeceleration,
	Jerk			:= MoveJerk,
	BufferMode     := MC_BlendingHigh,
	Axis			:= Master.Axis
);

Master.fbMC_MoveRelative[2](
	Execute  		:= FALSE,
	Axis			:= Master.Axis
);

END_FUNCTION_BLOCK

// ---- POUs/FB/SetMotionFuction.TcPOU
FUNCTION_BLOCK SetMotionFuction
VAR_INPUT
END_VAR
VAR_OUTPUT
END_VAR
VAR
	idx 				: INT:=2;
	AxisRunIdx		: ARRAY [0..MAX_ARRAY] OF INT:=[100(0)];
	MFIdx			: ARRAY[1..No] OF INT:=[No(1)];
	SlavePos		: ARRAY[1..No] OF LREAL:=[No(0)];
	TableNum		: INT:=0;
	MasterRatio		: LREAL;
	SlaveRatio		: LREAL;
END_VAR

MasterRatio :=360.0/1048576.0/4.0;
FOR idx := 2 TO No DO
	WHILE AxisProduce[idx].Dist[AxisRunIdx[idx]] <> 0 DO
		(*起始位置*)
		IF (AxisRunIdx[idx] <> 0) AND (AxisProduce[idx].Start[AxisRunIdx[idx]] <> AxisProduce[idx].End[AxisRunIdx[idx]-1]) THEN
			Cam[idx].MotionFunction[MFIdx[idx]].PointIndex       		 := MFIdx[idx];
		    	Cam[idx].MotionFunction[MFIdx[idx]].FunctionType     	 := MOTIONFUNCTYPE_POLYNOM5_MM;
		    	Cam[idx].MotionFunction[MFIdx[idx]].PointType        		 := MOTIONPOINTTYPE_REST;
		    	Cam[idx].MotionFunction[MFIdx[idx]].RelIndexNextPoint   := 1;
		    	Cam[idx].MotionFunction[MFIdx[idx]].MasterPos       	 	 := AxisProduce[idx].Start[AxisRunIdx[idx]]*MasterRatio;
		    	Cam[idx].MotionFunction[MFIdx[idx]].SlavePos         		 :=SlavePos[idx] ;
			MFIdx[idx]										 := MFIdx[idx] +1;
		ELSIF AxisRunIdx[idx] = 0 THEN
			(*主軸0度跟隨也在0度開始*)
			Cam[idx].MotionFunction[MFIdx[idx]].PointIndex       		 := MFIdx[idx];
		    	Cam[idx].MotionFunction[MFIdx[idx]].FunctionType     	 := MOTIONFUNCTYPE_POLYNOM5_MM;
		    	Cam[idx].MotionFunction[MFIdx[idx]].PointType        		 := MOTIONPOINTTYPE_REST;
		    	Cam[idx].MotionFunction[MFIdx[idx]].RelIndexNextPoint   := 1;
		    	Cam[idx].MotionFunction[MFIdx[idx]].MasterPos       	 	 :=0;
		    	Cam[idx].MotionFunction[MFIdx[idx]].SlavePos         		 :=0 ;
			MFIdx[idx]										 := MFIdx[idx] +1;

			Cam[idx].MotionFunction[MFIdx[idx]].PointIndex       		 := MFIdx[idx];
		    	Cam[idx].MotionFunction[MFIdx[idx]].FunctionType     	 := MOTIONFUNCTYPE_POLYNOM5_MM;
		    	Cam[idx].MotionFunction[MFIdx[idx]].PointType        		 := MOTIONPOINTTYPE_REST;
		    	Cam[idx].MotionFunction[MFIdx[idx]].RelIndexNextPoint   := 1;
		    	Cam[idx].MotionFunction[MFIdx[idx]].MasterPos       	 	 := AxisProduce[idx].Start[AxisRunIdx[idx]]*MasterRatio;
		    	Cam[idx].MotionFunction[MFIdx[idx]].SlavePos         		 :=SlavePos[idx] ;
			MFIdx[idx]										 := MFIdx[idx] +1;
		END_IF
		SlavePos[idx]									 := SlavePos[idx] + AxisProduce[idx].Dist[AxisRunIdx[idx]] ;
		(*結束位置*)
		Cam[idx].MotionFunction[MFIdx[idx]].PointIndex       		 := MFIdx[idx];
	    	Cam[idx].MotionFunction[MFIdx[idx]].FunctionType     	 := MOTIONFUNCTYPE_POLYNOM5_MM;
	    	Cam[idx].MotionFunction[MFIdx[idx]].PointType        		 := MOTIONPOINTTYPE_REST;
	    	Cam[idx].MotionFunction[MFIdx[idx]].RelIndexNextPoint   := 1;
	    	Cam[idx].MotionFunction[MFIdx[idx]].MasterPos       	 	 := AxisProduce[idx].End[AxisRunIdx[idx]]*MasterRatio;
	    	Cam[idx].MotionFunction[MFIdx[idx]].SlavePos         		 :=SlavePos[idx] ;

		MFIdx[idx]										 := MFIdx[idx] +1;
		AxisRunIdx[idx]									 := AxisRunIdx[idx] + 1;
	END_WHILE

	(*不是在360度結束*)
	IF Cam[idx].MotionFunction[MFIdx[idx]].MasterPos <360 THEN
		Cam[idx].MotionFunction[MFIdx[idx]].PointIndex       		 := MFIdx[idx];
	    	Cam[idx].MotionFunction[MFIdx[idx]].FunctionType     	 := MOTIONFUNCTYPE_POLYNOM5_MM;
	    	Cam[idx].MotionFunction[MFIdx[idx]].PointType        		 := MOTIONPOINTTYPE_REST;
	    	Cam[idx].MotionFunction[MFIdx[idx]].RelIndexNextPoint   := 0;
	    	Cam[idx].MotionFunction[MFIdx[idx]].MasterPos       	 	 := 360;
	    	Cam[idx].MotionFunction[MFIdx[idx]].SlavePos         		 := 0 ;
		MFIdx[idx]										 := MFIdx[idx] +1;
	END_IF


	AxisRunIdx[idx] 										 := AxisRunIdx[idx] - 1;
	MFIdx[idx]											 := MFIdx[idx] - 1;
	Cam[idx].MotionFunction[MFIdx[idx]].RelIndexNextPoint  		 := 0;(*最後的下一個點設0*)

	Cam[idx].Table.pArray			:= ADR( Cam[idx].MotionFunction );
	Cam[idx].Table.ArraySize		:= SIZEOF(Cam[idx].MotionFunction );
	Cam[idx].Table.TableType 		:= MC_TABLETYPE_MOTIONFUNCTION;
	Cam[idx].Table.NoOfRows		:= MFIdx[idx];
	Cam[idx].Table.NoOfColumns	:= 1;


END_FOR

END_FUNCTION_BLOCK

// ---- POUs/FB/SetPositionTable.TcPOU
FUNCTION_BLOCK SetPositionTable
VAR_INPUT
END_VAR
VAR_OUTPUT
END_VAR
VAR
	idx 				: INT:=2;
END_VAR



FOR idx := 1 TO No DO
	Cam[idx].Table.pArray			:= ADR( CamTable1[idx].PositionTable );
	Cam[idx].Table.ArraySize		:= SIZEOF(CamTable1[idx].PositionTable );
	Cam[idx].Table.TableType	 	:= MC_TABLETYPE_EQUIDISTANT;
	Cam[idx].Table.NoOfRows		:= CamTable1[idx].NoOfRows;
	Cam[idx].Table.NoOfColumns	:= 2;

	Cam[idx].Table2.pArray		:= ADR( CamTable2[idx].PositionTable );
	Cam[idx].Table2.ArraySize		:= SIZEOF(CamTable2[idx].PositionTable );
	Cam[idx].Table2.TableType 	:= MC_TABLETYPE_EQUIDISTANT;
	Cam[idx].Table2.NoOfRows		:= CamTable2[idx].NoOfRows;
	Cam[idx].Table2.NoOfColumns	:= 2;

END_FOR

END_FUNCTION_BLOCK
